ABB RAPID module: 76182c52.mod

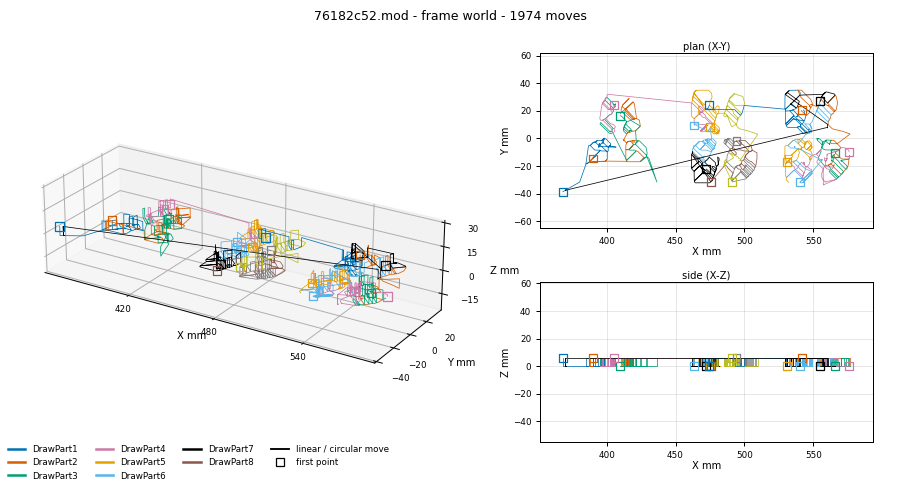
[picture p0: tool path of 76182c52.mod in frame world, 1974 of 1976 moves have a stored position in this frame; points joined in program order, loops and branches not executed]
MODULE ImageDraw
  ! Generated 2026-10-07 06:11 for ABB GoFa CRB 15000-5/0.95: 181 strokes
  ! Page 250 x 180 mm. Work object wPaper: Z points up, so pen-up is +Z and the tool uses orientation [0,1,0,0].
  PERS tooldata tPen:=[TRUE,[[0,0,120],[1,0,0,0]],[0.3,[0,0,60],[1,0,0,0],0,0,0]];
  PERS wobjdata wPaper:=[FALSE,TRUE,"",[[350,-90,0],[1,0,0,0]],[[0,0,0],[1,0,0,0]]];
  CONST robtarget pOrigin:=[[0,0,0],[0,1,0,0],[0,0,0,0],[9E9,9E9,9E9,9E9,9E9,9E9]];
  CONST jointtarget jHome:=[[0,0,0,0,30,0],[9E9,9E9,9E9,9E9,9E9,9E9]];
  CONST speeddata vTravel:=[250,200,5000,1000];

  PROC main()
    SingArea\Wrist;
    ConfL\Off;
    ConfJ\Off;
    MoveAbsJ jHome\NoEOffs,vTravel,fine,tPen;
    DrawPart1;
    DrawPart2;
    DrawPart3;
    DrawPart4;
    DrawPart5;
    DrawPart6;
    DrawPart7;
    DrawPart8;
    DrawPart9;
    DrawPart10;
    DrawPart11;
    DrawPart12;
    DrawPart13;
    DrawPart14;
    DrawPart15;
    DrawPart16;
    DrawPart17;
    MoveAbsJ jHome\NoEOffs,vTravel,fine,tPen;
  ENDPROC

  PROC DrawPart1()
    MoveL Offs(pOrigin,18.35,51.38,6.00),vTravel,z5,tPen\WObj:=wPaper;
    MoveL Offs(pOrigin,18.35,51.38,0.00),v60,z0,tPen\WObj:=wPaper;
    MoveL Offs(pOrigin,30.50,58.42,0.00),v40,z0,tPen\WObj:=wPaper;
    MoveL Offs(pOrigin,35.05,71.47,0.00),v40,z0,tPen\WObj:=wPaper;
    MoveL Offs(pOrigin,37.10,72.53,0.00),v40,z0,tPen\WObj:=wPaper;
    MoveL Offs(pOrigin,37.10,72.53,0.00),v40,z0,tPen\WObj:=wPaper;
    MoveL Offs(pOrigin,38.15,72.53,0.00),v40,z0,tPen\WObj:=wPaper;
    MoveL Offs(pOrigin,39.50,73.12,0.00),v40,z0,tPen\WObj:=wPaper;
    MoveL Offs(pOrigin,48.95,73.28,0.00),v40,z0,tPen\WObj:=wPaper;
    MoveL Offs(pOrigin,50.45,75.07,0.00),v40,z0,tPen\WObj:=wPaper;
    MoveL Offs(pOrigin,50.45,80.03,0.00),v40,z0,tPen\WObj:=wPaper;
    MoveL Offs(pOrigin,51.20,81.07,0.00),v40,z0,tPen\WObj:=wPaper;
    MoveL Offs(pOrigin,51.20,83.47,0.00),v40,z0,tPen\WObj:=wPaper;
    MoveL Offs(pOrigin,51.20,83.47,0.00),v40,z0,tPen\WObj:=wPaper;
    MoveL Offs(pOrigin,47.75,86.78,0.00),v40,z0,tPen\WObj:=wPaper;
    MoveL Offs(pOrigin,47.75,86.78,0.00),v40,z0,tPen\WObj:=wPaper;
    MoveL Offs(pOrigin,47.15,87.53,0.00),v40,z0,tPen\WObj:=wPaper;
    MoveL Offs(pOrigin,47.15,88.43,0.00),v40,z0,tPen\WObj:=wPaper;
    MoveL Offs(pOrigin,47.15,88.43,0.00),v40,z0,tPen\WObj:=wPaper;
    MoveL Offs(pOrigin,48.65,89.93,0.00),v40,z0,tPen\WObj:=wPaper;
    MoveL Offs(pOrigin,48.65,89.93,0.00),v40,z0,tPen\WObj:=wPaper;
    MoveL Offs(pOrigin,47.15,88.43,0.00),v40,z0,tPen\WObj:=wPaper;
    MoveL Offs(pOrigin,46.55,88.57,0.00),v40,z0,tPen\WObj:=wPaper;
    MoveL Offs(pOrigin,48.05,90.07,0.00),v40,fine,tPen\WObj:=wPaper;
    MoveL Offs(pOrigin,48.05,90.07,6.00),v60,z5,tPen\WObj:=wPaper;
    MoveL Offs(pOrigin,47.75,86.78,6.00),vTravel,z5,tPen\WObj:=wPaper;
    MoveL Offs(pOrigin,47.75,86.78,0.00),v60,z0,tPen\WObj:=wPaper;
    MoveL Offs(pOrigin,46.70,86.78,0.00),v40,z0,tPen\WObj:=wPaper;
    MoveL Offs(pOrigin,47.00,86.78,0.00),v40,fine,tPen\WObj:=wPaper;
    MoveL Offs(pOrigin,47.00,86.78,6.00),v60,z5,tPen\WObj:=wPaper;
    MoveL Offs(pOrigin,45.35,85.72,6.00),vTravel,z5,tPen\WObj:=wPaper;
    MoveL Offs(pOrigin,45.35,85.72,0.00),v60,z0,tPen\WObj:=wPaper;
    MoveL Offs(pOrigin,45.35,85.12,0.00),v40,z0,tPen\WObj:=wPaper;
    MoveL Offs(pOrigin,50.45,80.32,0.00),v40,z0,tPen\WObj:=wPaper;
    MoveL Offs(pOrigin,49.55,80.93,0.00),v40,z0,tPen\WObj:=wPaper;
    MoveL Offs(pOrigin,46.55,80.93,0.00),v40,z0,tPen\WObj:=wPaper;
    MoveL Offs(pOrigin,45.35,81.22,0.00),v40,z0,tPen\WObj:=wPaper;
    MoveL Offs(pOrigin,45.35,81.22,0.00),v40,z0,tPen\WObj:=wPaper;
    MoveL Offs(pOrigin,43.10,78.97,0.00),v40,z0,tPen\WObj:=wPaper;
    MoveL Offs(pOrigin,43.10,78.97,0.00),v40,z0,tPen\WObj:=wPaper;
    MoveL Offs(pOrigin,45.35,81.22,0.00),v40,z0,tPen\WObj:=wPaper;
    MoveL Offs(pOrigin,45.35,81.22,0.00),v40,z0,tPen\WObj:=wPaper;
    MoveL Offs(pOrigin,44.75,81.53,0.00),v40,z0,tPen\WObj:=wPaper;
    MoveL Offs(pOrigin,41.45,81.57,0.00),v40,z0,tPen\WObj:=wPaper;
    MoveL Offs(pOrigin,38.15,84.82,0.00),v40,z0,tPen\WObj:=wPaper;
    MoveL Offs(pOrigin,38.15,84.82,0.00),v40,z0,tPen\WObj:=wPaper;
    MoveL Offs(pOrigin,40.55,87.18,0.00),v40,z0,tPen\WObj:=wPaper;
    MoveL Offs(pOrigin,42.05,87.22,0.00),v40,z0,tPen\WObj:=wPaper;
    MoveL Offs(pOrigin,42.05,87.22,0.00),v40,z0,tPen\WObj:=wPaper;
    MoveL Offs(pOrigin,43.40,88.68,0.00),v40,z0,tPen\WObj:=wPaper;
    MoveL Offs(pOrigin,46.25,88.57,0.00),v40,z0,tPen\WObj:=wPaper;
    MoveL Offs(pOrigin,48.35,90.22,0.00),v40,z0,tPen\WObj:=wPaper;
    MoveL Offs(pOrigin,49.55,89.62,0.00),v40,z0,tPen\WObj:=wPaper;
    MoveL Offs(pOrigin,52.85,86.32,0.00),v40,z0,tPen\WObj:=wPaper;
    MoveL Offs(pOrigin,52.85,86.32,0.00),v40,z0,tPen\WObj:=wPaper;
    MoveL Offs(pOrigin,52.80,85.28,0.00),v40,z0,tPen\WObj:=wPaper;
    MoveL Offs(pOrigin,51.20,83.47,0.00),v40,z0,tPen\WObj:=wPaper;
    MoveL Offs(pOrigin,51.65,83.78,0.00),v40,z0,tPen\WObj:=wPaper;
    MoveL Offs(pOrigin,56.75,83.78,0.00),v40,z0,tPen\WObj:=wPaper;
    MoveL Offs(pOrigin,56.45,83.78,0.00),v40,fine,tPen\WObj:=wPaper;
    MoveL Offs(pOrigin,56.45,83.78,6.00),v60,z5,tPen\WObj:=wPaper;
    MoveL Offs(pOrigin,52.10,84.38,6.00),vTravel,z5,tPen\WObj:=wPaper;
    MoveL Offs(pOrigin,52.10,84.38,0.00),v60,z0,tPen\WObj:=wPaper;
    MoveL Offs(pOrigin,52.85,85.12,0.00),v40,z0,tPen\WObj:=wPaper;
    MoveL Offs(pOrigin,52.10,84.38,0.00),v40,fine,tPen\WObj:=wPaper;
    MoveL Offs(pOrigin,52.10,84.38,6.00),v60,z5,tPen\WObj:=wPaper;
    MoveL Offs(pOrigin,46.25,84.07,6.00),vTravel,z5,tPen\WObj:=wPaper;
    MoveL Offs(pOrigin,46.25,84.07,0.00),v60,z0,tPen\WObj:=wPaper;
    MoveL Offs(pOrigin,44.45,84.07,0.00),v40,z0,tPen\WObj:=wPaper;
    MoveL Offs(pOrigin,44.45,84.07,0.00),v40,z0,tPen\WObj:=wPaper;
    MoveL Offs(pOrigin,44.45,83.78,0.00),v40,z0,tPen\WObj:=wPaper;
    MoveL Offs(pOrigin,44.15,83.78,0.00),v40,z0,tPen\WObj:=wPaper;
    MoveL Offs(pOrigin,44.15,84.07,0.00),v40,z0,tPen\WObj:=wPaper;
    MoveL Offs(pOrigin,44.45,84.07,0.00),v40,z0,tPen\WObj:=wPaper;
    MoveL Offs(pOrigin,44.45,83.78,0.00),v40,z0,tPen\WObj:=wPaper;
    MoveL Offs(pOrigin,44.15,83.78,0.00),v40,z0,tPen\WObj:=wPaper;
    MoveL Offs(pOrigin,44.15,84.07,0.00),v40,z0,tPen\WObj:=wPaper;
    MoveL Offs(pOrigin,44.45,84.07,0.00),v40,z0,tPen\WObj:=wPaper;
    MoveL Offs(pOrigin,44.45,84.68,0.00),v40,z0,tPen\WObj:=wPaper;
    MoveL Offs(pOrigin,44.45,84.97,0.00),v40,z0,tPen\WObj:=wPaper;
    MoveL Offs(pOrigin,44.75,84.97,0.00),v40,z0,tPen\WObj:=wPaper;
    MoveL Offs(pOrigin,44.75,84.68,0.00),v40,z0,tPen\WObj:=wPaper;
    MoveL Offs(pOrigin,44.45,84.68,0.00),v40,z0,tPen\WObj:=wPaper;
    MoveL Offs(pOrigin,44.45,84.97,0.00),v40,z0,tPen\WObj:=wPaper;
    MoveL Offs(pOrigin,44.75,84.97,0.00),v40,z0,tPen\WObj:=wPaper;
    MoveL Offs(pOrigin,44.75,84.68,0.00),v40,z0,tPen\WObj:=wPaper;
    MoveL Offs(pOrigin,44.45,84.68,0.00),v40,z0,tPen\WObj:=wPaper;
    MoveL Offs(pOrigin,44.75,84.97,0.00),v40,z0,tPen\WObj:=wPaper;
    MoveL Offs(pOrigin,45.35,85.72,0.00),v40,z0,tPen\WObj:=wPaper;
    MoveL Offs(pOrigin,45.05,86.03,0.00),v40,z0,tPen\WObj:=wPaper;
    MoveL Offs(pOrigin,44.60,86.32,0.00),v40,z0,tPen\WObj:=wPaper;
    MoveL Offs(pOrigin,44.90,85.88,0.00),v40,z0,tPen\WObj:=wPaper;
    MoveL Offs(pOrigin,44.90,85.88,0.00),v40,z0,tPen\WObj:=wPaper;
    MoveL Offs(pOrigin,44.60,85.57,0.00),v40,z0,tPen\WObj:=wPaper;
    MoveL Offs(pOrigin,43.55,85.62,0.00),v40,z0,tPen\WObj:=wPaper;
    MoveL Offs(pOrigin,42.05,87.22,0.00),v40,z0,tPen\WObj:=wPaper;
    MoveL Offs(pOrigin,42.05,87.22,0.00),v40,z0,tPen\WObj:=wPaper;
    MoveL Offs(pOrigin,43.40,88.57,0.00),v40,fine,tPen\WObj:=wPaper;
    MoveL Offs(pOrigin,43.40,88.57,6.00),v60,z5,tPen\WObj:=wPaper;
    MoveL Offs(pOrigin,40.25,87.07,6.00),vTravel,z5,tPen\WObj:=wPaper;
    MoveL Offs(pOrigin,40.25,87.07,0.00),v60,z0,tPen\WObj:=wPaper;
    MoveL Offs(pOrigin,38.15,84.97,0.00),v40,z0,tPen\WObj:=wPaper;
    MoveL Offs(pOrigin,36.85,84.68,0.00),v40,z0,tPen\WObj:=wPaper;
    MoveL Offs(pOrigin,35.00,71.62,0.00),v40,fine,tPen\WObj:=wPaper;
    MoveL Offs(pOrigin,35.00,71.62,6.00),v60,z5,tPen\WObj:=wPaper;
    MoveL Offs(pOrigin,37.10,72.53,6.00),vTravel,z5,tPen\WObj:=wPaper;
    MoveL Offs(pOrigin,37.10,72.53,0.00),v60,z0,tPen\WObj:=wPaper;
    MoveL Offs(pOrigin,41.60,77.47,0.00),v40,z0,tPen\WObj:=wPaper;
    MoveL Offs(pOrigin,41.90,77.47,0.00),v40,z0,tPen\WObj:=wPaper;
    MoveL Offs(pOrigin,42.05,77.03,0.00),v40,z0,tPen\WObj:=wPaper;
    MoveL Offs(pOrigin,41.95,77.78,0.00),v40,z0,tPen\WObj:=wPaper;
    MoveL Offs(pOrigin,42.80,78.68,0.00),v40,z0,tPen\WObj:=wPaper;
    MoveL Offs(pOrigin,42.80,78.68,0.00),v40,z0,tPen\WObj:=wPaper;
    MoveL Offs(pOrigin,41.75,77.78,0.00),v40,z0,tPen\WObj:=wPaper;
    MoveL Offs(pOrigin,41.90,77.47,0.00),v40,fine,tPen\WObj:=wPaper;
    MoveL Offs(pOrigin,41.90,77.47,6.00),v60,z5,tPen\WObj:=wPaper;
    MoveL Offs(pOrigin,39.85,75.47,6.00),vTravel,z5,tPen\WObj:=wPaper;
    MoveL Offs(pOrigin,39.85,75.47,0.00),v60,z0,tPen\WObj:=wPaper;
    MoveL Offs(pOrigin,41.45,77.03,0.00),v40,z0,tPen\WObj:=wPaper;
    MoveL Offs(pOrigin,39.85,75.47,0.00),v40,fine,tPen\WObj:=wPaper;
  ENDPROC

  PROC DrawPart2()
    MoveL Offs(pOrigin,39.85,75.47,6.00),v60,z5,tPen\WObj:=wPaper;
    MoveL Offs(pOrigin,38.05,73.68,6.00),vTravel,z5,tPen\WObj:=wPaper;
    MoveL Offs(pOrigin,38.05,73.68,0.00),v60,z0,tPen\WObj:=wPaper;
    MoveL Offs(pOrigin,39.50,75.07,0.00),v40,z0,tPen\WObj:=wPaper;
    MoveL Offs(pOrigin,38.05,73.68,0.00),v40,z0,tPen\WObj:=wPaper;
    MoveL Offs(pOrigin,37.40,72.97,0.00),v40,z0,tPen\WObj:=wPaper;
    MoveL Offs(pOrigin,37.85,73.43,0.00),v40,z0,tPen\WObj:=wPaper;
    MoveL Offs(pOrigin,37.40,72.97,0.00),v40,fine,tPen\WObj:=wPaper;
    MoveL Offs(pOrigin,37.40,72.97,6.00),v60,z5,tPen\WObj:=wPaper;
    MoveL Offs(pOrigin,49.10,73.57,6.00),vTravel,z5,tPen\WObj:=wPaper;
    MoveL Offs(pOrigin,49.10,73.57,0.00),v60,z0,tPen\WObj:=wPaper;
    MoveL Offs(pOrigin,50.15,74.62,0.00),v40,z0,tPen\WObj:=wPaper;
    MoveL Offs(pOrigin,49.10,73.57,0.00),v40,fine,tPen\WObj:=wPaper;
    MoveL Offs(pOrigin,49.10,73.57,6.00),v60,z5,tPen\WObj:=wPaper;
    MoveL Offs(pOrigin,64.55,73.43,6.00),vTravel,z5,tPen\WObj:=wPaper;
    MoveL Offs(pOrigin,64.55,73.43,0.00),v60,z0,tPen\WObj:=wPaper;
    MoveL Offs(pOrigin,64.85,73.12,0.00),v40,z0,tPen\WObj:=wPaper;
    MoveL Offs(pOrigin,74.15,73.12,0.00),v40,z0,tPen\WObj:=wPaper;
    MoveL Offs(pOrigin,77.10,76.12,0.00),v40,z0,tPen\WObj:=wPaper;
    MoveL Offs(pOrigin,72.50,80.78,0.00),v40,z0,tPen\WObj:=wPaper;
    MoveL Offs(pOrigin,71.60,80.93,0.00),v40,z0,tPen\WObj:=wPaper;
    MoveL Offs(pOrigin,64.70,74.18,0.00),v40,z0,tPen\WObj:=wPaper;
    MoveL Offs(pOrigin,64.55,73.43,0.00),v40,z0,tPen\WObj:=wPaper;
    MoveL Offs(pOrigin,64.55,74.18,0.00),v40,z0,tPen\WObj:=wPaper;
    MoveL Offs(pOrigin,63.95,74.78,0.00),v40,z0,tPen\WObj:=wPaper;
    MoveL Offs(pOrigin,63.95,81.82,0.00),v40,fine,tPen\WObj:=wPaper;
    MoveL Offs(pOrigin,63.95,81.82,6.00),v60,z5,tPen\WObj:=wPaper;
    MoveL Offs(pOrigin,66.20,81.82,6.00),vTravel,z5,tPen\WObj:=wPaper;
    MoveL Offs(pOrigin,66.20,81.82,0.00),v60,z0,tPen\WObj:=wPaper;
    MoveL Offs(pOrigin,68.60,84.22,0.00),v40,fine,tPen\WObj:=wPaper;
    MoveL Offs(pOrigin,68.60,84.22,6.00),v60,z5,tPen\WObj:=wPaper;
    MoveL Offs(pOrigin,69.50,85.57,6.00),vTravel,z5,tPen\WObj:=wPaper;
    MoveL Offs(pOrigin,69.50,85.57,0.00),v60,z0,tPen\WObj:=wPaper;
    MoveL Offs(pOrigin,66.20,81.97,0.00),v40,z0,tPen\WObj:=wPaper;
    MoveL Offs(pOrigin,64.25,81.82,0.00),v40,z0,tPen\WObj:=wPaper;
    MoveL Offs(pOrigin,63.95,82.12,0.00),v40,z0,tPen\WObj:=wPaper;
    MoveL Offs(pOrigin,63.95,85.28,0.00),v40,z0,tPen\WObj:=wPaper;
    MoveL Offs(pOrigin,64.40,86.03,0.00),v40,z0,tPen\WObj:=wPaper;
    MoveL Offs(pOrigin,64.40,86.78,0.00),v40,z0,tPen\WObj:=wPaper;
    MoveL Offs(pOrigin,64.40,86.78,0.00),v40,z0,tPen\WObj:=wPaper;
    MoveL Offs(pOrigin,65.45,87.78,0.00),v40,z0,tPen\WObj:=wPaper;
    MoveL Offs(pOrigin,69.35,88.57,0.00),v40,z0,tPen\WObj:=wPaper;
    MoveL Offs(pOrigin,69.35,88.57,0.00),v40,z0,tPen\WObj:=wPaper;
    MoveL Offs(pOrigin,70.55,87.22,0.00),v40,z0,tPen\WObj:=wPaper;
    MoveL Offs(pOrigin,71.00,86.18,0.00),v40,z0,tPen\WObj:=wPaper;
    MoveL Offs(pOrigin,71.00,86.18,0.00),v40,z0,tPen\WObj:=wPaper;
    MoveL Offs(pOrigin,73.10,88.43,0.00),v40,z0,tPen\WObj:=wPaper;
    MoveL Offs(pOrigin,73.10,88.43,0.00),v40,z0,tPen\WObj:=wPaper;
    MoveL Offs(pOrigin,71.30,88.72,0.00),v40,z0,tPen\WObj:=wPaper;
    MoveL Offs(pOrigin,69.35,88.57,0.00),v40,z0,tPen\WObj:=wPaper;
    MoveL Offs(pOrigin,68.60,88.28,0.00),v40,z0,tPen\WObj:=wPaper;
    MoveL Offs(pOrigin,69.20,87.53,0.00),v40,fine,tPen\WObj:=wPaper;
    MoveL Offs(pOrigin,69.20,87.53,6.00),v60,z5,tPen\WObj:=wPaper;
    MoveL Offs(pOrigin,69.20,86.03,6.00),vTravel,z5,tPen\WObj:=wPaper;
    MoveL Offs(pOrigin,69.20,86.03,0.00),v60,z0,tPen\WObj:=wPaper;
    MoveL Offs(pOrigin,67.55,87.97,0.00),v40,fine,tPen\WObj:=wPaper;
    MoveL Offs(pOrigin,67.55,87.97,6.00),v60,z5,tPen\WObj:=wPaper;
    MoveL Offs(pOrigin,65.45,87.68,6.00),vTravel,z5,tPen\WObj:=wPaper;
    MoveL Offs(pOrigin,65.45,87.68,0.00),v60,z0,tPen\WObj:=wPaper;
    MoveL Offs(pOrigin,64.40,86.78,0.00),v40,z0,tPen\WObj:=wPaper;
    MoveL Offs(pOrigin,64.40,86.78,0.00),v40,z0,tPen\WObj:=wPaper;
    MoveL Offs(pOrigin,62.75,88.43,0.00),v40,z0,tPen\WObj:=wPaper;
    MoveL Offs(pOrigin,62.00,89.03,0.00),v40,z0,tPen\WObj:=wPaper;
    MoveL Offs(pOrigin,62.70,88.57,0.00),v40,z0,tPen\WObj:=wPaper;
    MoveL Offs(pOrigin,62.75,89.78,0.00),v40,fine,tPen\WObj:=wPaper;
    MoveL Offs(pOrigin,62.75,89.78,6.00),v60,z5,tPen\WObj:=wPaper;
    MoveL Offs(pOrigin,65.15,94.12,6.00),vTravel,z5,tPen\WObj:=wPaper;
    MoveL Offs(pOrigin,65.15,94.12,0.00),v60,z0,tPen\WObj:=wPaper;
    MoveL Offs(pOrigin,65.60,94.72,0.00),v40,z0,tPen\WObj:=wPaper;
    MoveL Offs(pOrigin,66.05,94.12,0.00),v40,z0,tPen\WObj:=wPaper;
    MoveL Offs(pOrigin,66.05,94.12,0.00),v40,z0,tPen\WObj:=wPaper;
    MoveL Offs(pOrigin,68.90,95.32,0.00),v40,z0,tPen\WObj:=wPaper;
    MoveL Offs(pOrigin,70.85,95.43,0.00),v40,z0,tPen\WObj:=wPaper;
    MoveL Offs(pOrigin,74.45,98.93,0.00),v40,z0,tPen\WObj:=wPaper;
    MoveL Offs(pOrigin,74.45,98.93,0.00),v40,z0,tPen\WObj:=wPaper;
    MoveL Offs(pOrigin,73.80,103.28,0.00),v40,z0,tPen\WObj:=wPaper;
    MoveL Offs(pOrigin,71.60,104.47,0.00),v40,z0,tPen\WObj:=wPaper;
    MoveL Offs(pOrigin,70.70,104.32,0.00),v40,z0,tPen\WObj:=wPaper;
    MoveL Offs(pOrigin,69.80,104.03,0.00),v40,z0,tPen\WObj:=wPaper;
    MoveL Offs(pOrigin,69.80,104.03,0.00),v40,z0,tPen\WObj:=wPaper;
    MoveL Offs(pOrigin,68.60,104.03,0.00),v40,z0,tPen\WObj:=wPaper;
    MoveL Offs(pOrigin,63.20,109.57,0.00),v40,z0,tPen\WObj:=wPaper;
    MoveL Offs(pOrigin,63.20,109.57,0.00),v40,z0,tPen\WObj:=wPaper;
    MoveL Offs(pOrigin,63.80,110.47,0.00),v40,z0,tPen\WObj:=wPaper;
    MoveL Offs(pOrigin,63.80,110.47,0.00),v40,z0,tPen\WObj:=wPaper;
    MoveL Offs(pOrigin,69.80,104.03,0.00),v40,z0,tPen\WObj:=wPaper;
    MoveL Offs(pOrigin,70.70,104.32,0.00),v40,z0,tPen\WObj:=wPaper;
    MoveL Offs(pOrigin,65.30,109.88,0.00),v40,fine,tPen\WObj:=wPaper;
    MoveL Offs(pOrigin,65.30,109.88,6.00),v60,z5,tPen\WObj:=wPaper;
    MoveL Offs(pOrigin,64.10,111.53,6.00),vTravel,z5,tPen\WObj:=wPaper;
    MoveL Offs(pOrigin,64.10,111.53,0.00),v60,z0,tPen\WObj:=wPaper;
    MoveL Offs(pOrigin,69.20,116.47,0.00),v40,z0,tPen\WObj:=wPaper;
    MoveL Offs(pOrigin,69.20,116.47,0.00),v40,z0,tPen\WObj:=wPaper;
    MoveL Offs(pOrigin,70.10,115.28,0.00),v40,z0,tPen\WObj:=wPaper;
    MoveL Offs(pOrigin,71.60,105.38,0.00),v40,z0,tPen\WObj:=wPaper;
    MoveL Offs(pOrigin,71.45,104.47,0.00),v40,z0,tPen\WObj:=wPaper;
    MoveL Offs(pOrigin,70.70,104.32,0.00),v40,fine,tPen\WObj:=wPaper;
    MoveL Offs(pOrigin,70.70,104.32,6.00),v60,z5,tPen\WObj:=wPaper;
    MoveL Offs(pOrigin,68.60,103.88,6.00),vTravel,z5,tPen\WObj:=wPaper;
    MoveL Offs(pOrigin,68.60,103.88,0.00),v60,z0,tPen\WObj:=wPaper;
    MoveL Offs(pOrigin,68.00,103.32,0.00),v40,z0,tPen\WObj:=wPaper;
    MoveL Offs(pOrigin,67.40,103.43,0.00),v40,z0,tPen\WObj:=wPaper;
    MoveL Offs(pOrigin,60.50,110.03,0.00),v40,z0,tPen\WObj:=wPaper;
    MoveL Offs(pOrigin,60.50,110.03,0.00),v40,z0,tPen\WObj:=wPaper;
    MoveL Offs(pOrigin,60.65,111.68,0.00),v40,z0,tPen\WObj:=wPaper;
    MoveL Offs(pOrigin,61.60,114.22,0.00),v40,z0,tPen\WObj:=wPaper;
    MoveL Offs(pOrigin,66.35,119.03,0.00),v40,z0,tPen\WObj:=wPaper;
    MoveL Offs(pOrigin,66.35,119.03,0.00),v40,z0,tPen\WObj:=wPaper;
    MoveL Offs(pOrigin,61.70,114.22,0.00),v40,fine,tPen\WObj:=wPaper;
    MoveL Offs(pOrigin,61.70,114.22,6.00),v60,z5,tPen\WObj:=wPaper;
    MoveL Offs(pOrigin,61.40,112.88,6.00),vTravel,z5,tPen\WObj:=wPaper;
    MoveL Offs(pOrigin,61.40,112.88,0.00),v60,z0,tPen\WObj:=wPaper;
    MoveL Offs(pOrigin,63.50,111.22,0.00),v40,z0,tPen\WObj:=wPaper;
    MoveL Offs(pOrigin,63.50,111.22,0.00),v40,z0,tPen\WObj:=wPaper;
    MoveL Offs(pOrigin,64.25,111.53,0.00),v40,z0,tPen\WObj:=wPaper;
    MoveL Offs(pOrigin,69.20,116.47,0.00),v40,fine,tPen\WObj:=wPaper;
    MoveL Offs(pOrigin,69.20,116.47,6.00),v60,z5,tPen\WObj:=wPaper;
    MoveL Offs(pOrigin,60.50,108.53,6.00),vTravel,z5,tPen\WObj:=wPaper;
    MoveL Offs(pOrigin,60.50,108.53,0.00),v60,z0,tPen\WObj:=wPaper;
    MoveL Offs(pOrigin,59.90,107.93,0.00),v40,z0,tPen\WObj:=wPaper;
  ENDPROC

  PROC DrawPart3()
    MoveL Offs(pOrigin,59.90,106.57,0.00),v40,z0,tPen\WObj:=wPaper;
    MoveL Offs(pOrigin,59.90,106.57,0.00),v40,z0,tPen\WObj:=wPaper;
    MoveL Offs(pOrigin,60.65,106.28,0.00),v40,z0,tPen\WObj:=wPaper;
    MoveL Offs(pOrigin,64.55,102.38,0.00),v40,z0,tPen\WObj:=wPaper;
    MoveL Offs(pOrigin,64.55,102.38,0.00),v40,z0,tPen\WObj:=wPaper;
    MoveL Offs(pOrigin,63.90,100.43,0.00),v40,z0,tPen\WObj:=wPaper;
    MoveL Offs(pOrigin,62.95,99.38,0.00),v40,z0,tPen\WObj:=wPaper;
    MoveL Offs(pOrigin,62.50,98.18,0.00),v40,z0,tPen\WObj:=wPaper;
    MoveL Offs(pOrigin,62.15,95.62,0.00),v40,z0,tPen\WObj:=wPaper;
    MoveL Offs(pOrigin,64.10,93.57,0.00),v40,z0,tPen\WObj:=wPaper;
    MoveL Offs(pOrigin,64.80,93.57,0.00),v40,z0,tPen\WObj:=wPaper;
    MoveL Offs(pOrigin,65.15,94.12,0.00),v40,z0,tPen\WObj:=wPaper;
    MoveL Offs(pOrigin,65.30,94.28,0.00),v40,z0,tPen\WObj:=wPaper;
    MoveL Offs(pOrigin,62.45,96.97,0.00),v40,fine,tPen\WObj:=wPaper;
    MoveL Offs(pOrigin,62.45,96.97,6.00),v60,z5,tPen\WObj:=wPaper;
    MoveL Offs(pOrigin,62.90,98.47,6.00),vTravel,z5,tPen\WObj:=wPaper;
    MoveL Offs(pOrigin,62.90,98.47,0.00),v60,z0,tPen\WObj:=wPaper;
    MoveL Offs(pOrigin,66.80,94.43,0.00),v40,fine,tPen\WObj:=wPaper;
    MoveL Offs(pOrigin,66.80,94.43,6.00),v60,z5,tPen\WObj:=wPaper;
    MoveL Offs(pOrigin,66.65,95.62,6.00),vTravel,z5,tPen\WObj:=wPaper;
    MoveL Offs(pOrigin,66.65,95.62,0.00),v60,z0,tPen\WObj:=wPaper;
    MoveL Offs(pOrigin,66.80,95.32,0.00),v40,z0,tPen\WObj:=wPaper;
    MoveL Offs(pOrigin,67.10,95.47,0.00),v40,z0,tPen\WObj:=wPaper;
    MoveL Offs(pOrigin,66.80,95.78,0.00),v40,fine,tPen\WObj:=wPaper;
    MoveL Offs(pOrigin,66.80,95.78,6.00),v60,z5,tPen\WObj:=wPaper;
    MoveL Offs(pOrigin,68.60,95.32,6.00),vTravel,z5,tPen\WObj:=wPaper;
    MoveL Offs(pOrigin,68.60,95.32,0.00),v60,z0,tPen\WObj:=wPaper;
    MoveL Offs(pOrigin,67.25,97.12,0.00),v40,z0,tPen\WObj:=wPaper;
    MoveL Offs(pOrigin,63.95,100.28,0.00),v40,z0,tPen\WObj:=wPaper;
    MoveL Offs(pOrigin,63.95,100.28,0.00),v40,z0,tPen\WObj:=wPaper;
    MoveL Offs(pOrigin,63.05,99.38,0.00),v40,fine,tPen\WObj:=wPaper;
    MoveL Offs(pOrigin,63.05,99.38,6.00),v60,z5,tPen\WObj:=wPaper;
    MoveL Offs(pOrigin,64.55,102.38,6.00),vTravel,z5,tPen\WObj:=wPaper;
    MoveL Offs(pOrigin,64.55,102.38,0.00),v60,z0,tPen\WObj:=wPaper;
    MoveL Offs(pOrigin,65.60,102.38,0.00),v40,z0,tPen\WObj:=wPaper;
    MoveL Offs(pOrigin,67.40,103.28,0.00),v40,fine,tPen\WObj:=wPaper;
    MoveL Offs(pOrigin,67.40,103.28,6.00),v60,z5,tPen\WObj:=wPaper;
    MoveL Offs(pOrigin,74.45,98.93,6.00),vTravel,z5,tPen\WObj:=wPaper;
    MoveL Offs(pOrigin,74.45,98.93,0.00),v60,z0,tPen\WObj:=wPaper;
    MoveL Offs(pOrigin,71.00,95.62,0.00),v40,fine,tPen\WObj:=wPaper;
    MoveL Offs(pOrigin,71.00,95.62,6.00),v60,z5,tPen\WObj:=wPaper;
    MoveL Offs(pOrigin,71.60,86.78,6.00),vTravel,z5,tPen\WObj:=wPaper;
    MoveL Offs(pOrigin,71.60,86.78,0.00),v60,z0,tPen\WObj:=wPaper;
    MoveL Offs(pOrigin,73.10,88.28,0.00),v40,z0,tPen\WObj:=wPaper;
    MoveL Offs(pOrigin,73.70,88.38,0.00),v40,z0,tPen\WObj:=wPaper;
    MoveL Offs(pOrigin,78.65,83.47,0.00),v40,z0,tPen\WObj:=wPaper;
    MoveL Offs(pOrigin,79.40,79.43,0.00),v40,z0,tPen\WObj:=wPaper;
    MoveL Offs(pOrigin,79.35,78.53,0.00),v40,z0,tPen\WObj:=wPaper;
    MoveL Offs(pOrigin,78.80,77.93,0.00),v40,z0,tPen\WObj:=wPaper;
    MoveL Offs(pOrigin,78.80,77.93,0.00),v40,z0,tPen\WObj:=wPaper;
    MoveL Offs(pOrigin,78.80,76.72,0.00),v40,z0,tPen\WObj:=wPaper;
    MoveL Offs(pOrigin,78.20,76.18,0.00),v40,z0,tPen\WObj:=wPaper;
    MoveL Offs(pOrigin,77.15,75.97,0.00),v40,z0,tPen\WObj:=wPaper;
    MoveL Offs(pOrigin,77.15,75.97,0.00),v40,z0,tPen\WObj:=wPaper;
    MoveL Offs(pOrigin,74.60,73.28,0.00),v40,fine,tPen\WObj:=wPaper;
    MoveL Offs(pOrigin,74.60,73.28,6.00),v60,z5,tPen\WObj:=wPaper;
    MoveL Offs(pOrigin,78.95,76.72,6.00),vTravel,z5,tPen\WObj:=wPaper;
    MoveL Offs(pOrigin,78.95,76.72,0.00),v60,z0,tPen\WObj:=wPaper;
    MoveL Offs(pOrigin,80.60,75.82,0.00),v40,z0,tPen\WObj:=wPaper;
    MoveL Offs(pOrigin,86.45,58.42,0.00),v40,fine,tPen\WObj:=wPaper;
    MoveL Offs(pOrigin,86.45,58.42,6.00),v60,z5,tPen\WObj:=wPaper;
    MoveL Offs(pOrigin,78.80,77.93,6.00),vTravel,z5,tPen\WObj:=wPaper;
    MoveL Offs(pOrigin,78.80,77.93,0.00),v60,z0,tPen\WObj:=wPaper;
    MoveL Offs(pOrigin,71.15,85.57,0.00),v40,z0,tPen\WObj:=wPaper;
    MoveL Offs(pOrigin,71.00,86.18,0.00),v40,z0,tPen\WObj:=wPaper;
    MoveL Offs(pOrigin,71.00,85.57,0.00),v40,z0,tPen\WObj:=wPaper;
    MoveL Offs(pOrigin,69.50,85.72,0.00),v40,fine,tPen\WObj:=wPaper;
    MoveL Offs(pOrigin,69.50,85.72,6.00),v60,z5,tPen\WObj:=wPaper;
    MoveL Offs(pOrigin,66.20,81.82,6.00),vTravel,z5,tPen\WObj:=wPaper;
    MoveL Offs(pOrigin,66.20,81.82,0.00),v60,z0,tPen\WObj:=wPaper;
    MoveL Offs(pOrigin,66.80,81.53,0.00),v40,z0,tPen\WObj:=wPaper;
    MoveL Offs(pOrigin,70.55,81.53,0.00),v40,z0,tPen\WObj:=wPaper;
    MoveL Offs(pOrigin,71.30,80.93,0.00),v40,z0,tPen\WObj:=wPaper;
    MoveL Offs(pOrigin,71.30,80.93,0.00),v40,z0,tPen\WObj:=wPaper;
    MoveL Offs(pOrigin,64.55,74.18,0.00),v40,fine,tPen\WObj:=wPaper;
    MoveL Offs(pOrigin,64.55,74.18,6.00),v60,z5,tPen\WObj:=wPaper;
    MoveL Offs(pOrigin,54.35,94.43,6.00),vTravel,z5,tPen\WObj:=wPaper;
    MoveL Offs(pOrigin,54.35,94.43,0.00),v60,z0,tPen\WObj:=wPaper;
    MoveL Offs(pOrigin,53.60,93.68,0.00),v40,z0,tPen\WObj:=wPaper;
    MoveL Offs(pOrigin,52.10,93.72,0.00),v40,z0,tPen\WObj:=wPaper;
    MoveL Offs(pOrigin,45.20,100.43,0.00),v40,fine,tPen\WObj:=wPaper;
    MoveL Offs(pOrigin,45.20,100.43,6.00),v60,z5,tPen\WObj:=wPaper;
    MoveL Offs(pOrigin,45.65,101.62,6.00),vTravel,z5,tPen\WObj:=wPaper;
    MoveL Offs(pOrigin,45.65,101.62,0.00),v60,z0,tPen\WObj:=wPaper;
    MoveL Offs(pOrigin,52.25,95.18,0.00),v40,z0,tPen\WObj:=wPaper;
    MoveL Offs(pOrigin,52.55,95.32,0.00),v40,z0,tPen\WObj:=wPaper;
    MoveL Offs(pOrigin,52.55,94.72,0.00),v40,z0,tPen\WObj:=wPaper;
    MoveL Offs(pOrigin,52.85,95.32,0.00),v40,z0,tPen\WObj:=wPaper;
    MoveL Offs(pOrigin,54.05,95.03,0.00),v40,z0,tPen\WObj:=wPaper;
    MoveL Offs(pOrigin,54.05,95.03,0.00),v40,z0,tPen\WObj:=wPaper;
    MoveL Offs(pOrigin,53.90,96.68,0.00),v40,z0,tPen\WObj:=wPaper;
    MoveL Offs(pOrigin,53.90,96.68,0.00),v40,z0,tPen\WObj:=wPaper;
    MoveL Offs(pOrigin,54.95,97.12,0.00),v40,z0,tPen\WObj:=wPaper;
    MoveL Offs(pOrigin,54.95,97.12,0.00),v40,z0,tPen\WObj:=wPaper;
    MoveL Offs(pOrigin,48.50,103.88,0.00),v40,z0,tPen\WObj:=wPaper;
    MoveL Offs(pOrigin,48.50,103.88,0.00),v40,z0,tPen\WObj:=wPaper;
    MoveL Offs(pOrigin,52.10,107.18,0.00),v40,fine,tPen\WObj:=wPaper;
    MoveL Offs(pOrigin,52.10,107.18,6.00),v60,z5,tPen\WObj:=wPaper;
    MoveL Offs(pOrigin,53.45,107.62,6.00),vTravel,z5,tPen\WObj:=wPaper;
    MoveL Offs(pOrigin,53.45,107.62,0.00),v60,z0,tPen\WObj:=wPaper;
    MoveL Offs(pOrigin,54.85,109.57,0.00),v40,z0,tPen\WObj:=wPaper;
    MoveL Offs(pOrigin,54.95,111.82,0.00),v40,z0,tPen\WObj:=wPaper;
    MoveL Offs(pOrigin,54.95,111.82,0.00),v40,z0,tPen\WObj:=wPaper;
    MoveL Offs(pOrigin,48.80,117.82,0.00),v40,z0,tPen\WObj:=wPaper;
    MoveL Offs(pOrigin,48.80,117.82,0.00),v40,z0,tPen\WObj:=wPaper;
    MoveL Offs(pOrigin,49.05,119.18,0.00),v40,z0,tPen\WObj:=wPaper;
    MoveL Offs(pOrigin,50.15,119.93,0.00),v40,z0,tPen\WObj:=wPaper;
    MoveL Offs(pOrigin,50.15,119.93,0.00),v40,z0,tPen\WObj:=wPaper;
    MoveL Offs(pOrigin,54.65,115.43,0.00),v40,z0,tPen\WObj:=wPaper;
    MoveL Offs(pOrigin,54.70,114.72,0.00),v40,z0,tPen\WObj:=wPaper;
    MoveL Offs(pOrigin,54.95,114.97,0.00),v40,z0,tPen\WObj:=wPaper;
    MoveL Offs(pOrigin,54.95,114.97,0.00),v40,z0,tPen\WObj:=wPaper;
    MoveL Offs(pOrigin,55.70,114.38,0.00),v40,z0,tPen\WObj:=wPaper;
    MoveL Offs(pOrigin,56.45,114.57,0.00),v40,z0,tPen\WObj:=wPaper;
    MoveL Offs(pOrigin,56.60,115.12,0.00),v40,z0,tPen\WObj:=wPaper;
    MoveL Offs(pOrigin,56.00,114.38,0.00),v40,z0,tPen\WObj:=wPaper;
    MoveL Offs(pOrigin,56.45,113.47,0.00),v40,z0,tPen\WObj:=wPaper;
    MoveL Offs(pOrigin,55.40,112.43,0.00),v40,z0,tPen\WObj:=wPaper;
    MoveL Offs(pOrigin,55.40,112.43,0.00),v40,z0,tPen\WObj:=wPaper;
    MoveL Offs(pOrigin,55.40,114.38,0.00),v40,fine,tPen\WObj:=wPaper;
  ENDPROC

  PROC DrawPart4()
    MoveL Offs(pOrigin,55.40,114.38,6.00),v60,z5,tPen\WObj:=wPaper;
    MoveL Offs(pOrigin,55.70,112.43,6.00),vTravel,z5,tPen\WObj:=wPaper;
    MoveL Offs(pOrigin,55.70,112.43,0.00),v60,z0,tPen\WObj:=wPaper;
    MoveL Offs(pOrigin,56.45,113.18,0.00),v40,z0,tPen\WObj:=wPaper;
    MoveL Offs(pOrigin,55.70,112.43,0.00),v40,fine,tPen\WObj:=wPaper;
    MoveL Offs(pOrigin,55.70,112.43,6.00),v60,z5,tPen\WObj:=wPaper;
    MoveL Offs(pOrigin,52.40,111.22,6.00),vTravel,z5,tPen\WObj:=wPaper;
    MoveL Offs(pOrigin,52.40,111.22,0.00),v60,z0,tPen\WObj:=wPaper;
    MoveL Offs(pOrigin,54.20,109.12,0.00),v40,fine,tPen\WObj:=wPaper;
    MoveL Offs(pOrigin,54.20,109.12,6.00),v60,z5,tPen\WObj:=wPaper;
    MoveL Offs(pOrigin,53.45,107.62,6.00),vTravel,z5,tPen\WObj:=wPaper;
    MoveL Offs(pOrigin,53.45,107.62,0.00),v60,z0,tPen\WObj:=wPaper;
    MoveL Offs(pOrigin,52.25,107.18,0.00),v40,z0,tPen\WObj:=wPaper;
    MoveL Offs(pOrigin,49.40,104.32,0.00),v40,z0,tPen\WObj:=wPaper;
    MoveL Offs(pOrigin,49.40,104.32,0.00),v40,z0,tPen\WObj:=wPaper;
    MoveL Offs(pOrigin,52.70,100.88,0.00),v40,z0,tPen\WObj:=wPaper;
    MoveL Offs(pOrigin,54.95,100.12,0.00),v40,z0,tPen\WObj:=wPaper;
    MoveL Offs(pOrigin,56.20,98.78,0.00),v40,z0,tPen\WObj:=wPaper;
    MoveL Offs(pOrigin,56.30,98.03,0.00),v40,z0,tPen\WObj:=wPaper;
    MoveL Offs(pOrigin,56.30,98.03,0.00),v40,z0,tPen\WObj:=wPaper;
    MoveL Offs(pOrigin,55.40,97.12,0.00),v40,z0,tPen\WObj:=wPaper;
    MoveL Offs(pOrigin,55.40,97.12,0.00),v40,z0,tPen\WObj:=wPaper;
    MoveL Offs(pOrigin,55.95,95.18,0.00),v40,z0,tPen\WObj:=wPaper;
    MoveL Offs(pOrigin,55.10,94.43,0.00),v40,z0,tPen\WObj:=wPaper;
    MoveL Offs(pOrigin,54.50,94.47,0.00),v40,z0,tPen\WObj:=wPaper;
    MoveL Offs(pOrigin,54.05,95.03,0.00),v40,fine,tPen\WObj:=wPaper;
    MoveL Offs(pOrigin,54.05,95.03,6.00),v60,z5,tPen\WObj:=wPaper;
    MoveL Offs(pOrigin,53.90,96.68,6.00),vTravel,z5,tPen\WObj:=wPaper;
    MoveL Offs(pOrigin,53.90,96.68,0.00),v60,z0,tPen\WObj:=wPaper;
    MoveL Offs(pOrigin,47.15,103.28,0.00),v40,z0,tPen\WObj:=wPaper;
    MoveL Offs(pOrigin,47.15,103.28,0.00),v40,z0,tPen\WObj:=wPaper;
    MoveL Offs(pOrigin,47.75,103.88,0.00),v40,z0,tPen\WObj:=wPaper;
    MoveL Offs(pOrigin,48.50,103.88,0.00),v40,fine,tPen\WObj:=wPaper;
    MoveL Offs(pOrigin,48.50,103.88,6.00),v60,z5,tPen\WObj:=wPaper;
    MoveL Offs(pOrigin,47.15,103.28,6.00),vTravel,z5,tPen\WObj:=wPaper;
    MoveL Offs(pOrigin,47.15,103.28,0.00),v60,z0,tPen\WObj:=wPaper;
    MoveL Offs(pOrigin,45.80,103.12,0.00),v40,z0,tPen\WObj:=wPaper;
    MoveL Offs(pOrigin,45.80,103.12,0.00),v40,z0,tPen\WObj:=wPaper;
    MoveL Offs(pOrigin,45.05,104.32,0.00),v40,z0,tPen\WObj:=wPaper;
    MoveL Offs(pOrigin,46.55,114.38,0.00),v40,z0,tPen\WObj:=wPaper;
    MoveL Offs(pOrigin,47.00,115.12,0.00),v40,z0,tPen\WObj:=wPaper;
    MoveL Offs(pOrigin,47.00,115.12,0.00),v40,z0,tPen\WObj:=wPaper;
    MoveL Offs(pOrigin,51.20,111.07,0.00),v40,z0,tPen\WObj:=wPaper;
    MoveL Offs(pOrigin,51.20,111.07,0.00),v40,z0,tPen\WObj:=wPaper;
    MoveL Offs(pOrigin,51.50,111.07,0.00),v40,z0,tPen\WObj:=wPaper;
    MoveL Offs(pOrigin,51.35,110.78,0.00),v40,z0,tPen\WObj:=wPaper;
    MoveL Offs(pOrigin,51.20,111.07,0.00),v40,z0,tPen\WObj:=wPaper;
    MoveL Offs(pOrigin,51.50,111.07,0.00),v40,z0,tPen\WObj:=wPaper;
    MoveL Offs(pOrigin,51.20,110.78,0.00),v40,z0,tPen\WObj:=wPaper;
    MoveL Offs(pOrigin,51.20,111.07,0.00),v40,fine,tPen\WObj:=wPaper;
    MoveL Offs(pOrigin,51.20,111.07,6.00),v60,z5,tPen\WObj:=wPaper;
    MoveL Offs(pOrigin,52.40,111.22,6.00),vTravel,z5,tPen\WObj:=wPaper;
    MoveL Offs(pOrigin,52.40,111.22,0.00),v60,z0,tPen\WObj:=wPaper;
    MoveL Offs(pOrigin,47.45,116.03,0.00),v40,z0,tPen\WObj:=wPaper;
    MoveL Offs(pOrigin,47.45,116.03,0.00),v40,z0,tPen\WObj:=wPaper;
    MoveL Offs(pOrigin,47.75,117.07,0.00),v40,z0,tPen\WObj:=wPaper;
    MoveL Offs(pOrigin,48.80,117.82,0.00),v40,fine,tPen\WObj:=wPaper;
    MoveL Offs(pOrigin,48.80,117.82,6.00),v60,z5,tPen\WObj:=wPaper;
    MoveL Offs(pOrigin,47.45,116.03,6.00),vTravel,z5,tPen\WObj:=wPaper;
    MoveL Offs(pOrigin,47.45,116.03,0.00),v60,z0,tPen\WObj:=wPaper;
    MoveL Offs(pOrigin,47.00,115.72,0.00),v40,z0,tPen\WObj:=wPaper;
    MoveL Offs(pOrigin,47.00,115.12,0.00),v40,fine,tPen\WObj:=wPaper;
    MoveL Offs(pOrigin,47.00,115.12,6.00),v60,z5,tPen\WObj:=wPaper;
    MoveL Offs(pOrigin,50.15,119.93,6.00),vTravel,z5,tPen\WObj:=wPaper;
    MoveL Offs(pOrigin,50.15,119.93,0.00),v60,z0,tPen\WObj:=wPaper;
    MoveL Offs(pOrigin,50.35,121.72,0.00),v40,z0,tPen\WObj:=wPaper;
    MoveL Offs(pOrigin,50.90,122.03,0.00),v40,fine,tPen\WObj:=wPaper;
    MoveL Offs(pOrigin,50.90,122.03,6.00),v60,z5,tPen\WObj:=wPaper;
    MoveL Offs(pOrigin,111.95,115.72,6.00),vTravel,z5,tPen\WObj:=wPaper;
    MoveL Offs(pOrigin,111.95,115.72,0.00),v60,z0,tPen\WObj:=wPaper;
    MoveL Offs(pOrigin,118.85,108.97,0.00),v40,z0,tPen\WObj:=wPaper;
    MoveL Offs(pOrigin,119.45,108.97,0.00),v40,z0,tPen\WObj:=wPaper;
    MoveL Offs(pOrigin,121.40,107.03,0.00),v40,z0,tPen\WObj:=wPaper;
    MoveL Offs(pOrigin,122.00,105.68,0.00),v40,z0,tPen\WObj:=wPaper;
    MoveL Offs(pOrigin,127.25,100.72,0.00),v40,z0,tPen\WObj:=wPaper;
    MoveL Offs(pOrigin,127.25,100.72,0.00),v40,z0,tPen\WObj:=wPaper;
    MoveL Offs(pOrigin,126.95,99.97,0.00),v40,z0,tPen\WObj:=wPaper;
    MoveL Offs(pOrigin,126.50,99.97,0.00),v40,z0,tPen\WObj:=wPaper;
    MoveL Offs(pOrigin,126.50,99.97,0.00),v40,z0,tPen\WObj:=wPaper;
    MoveL Offs(pOrigin,121.25,105.03,0.00),v40,z0,tPen\WObj:=wPaper;
    MoveL Offs(pOrigin,119.60,105.53,0.00),v40,z0,tPen\WObj:=wPaper;
    MoveL Offs(pOrigin,117.65,107.62,0.00),v40,z0,tPen\WObj:=wPaper;
    MoveL Offs(pOrigin,117.65,107.62,0.00),v40,z0,tPen\WObj:=wPaper;
    MoveL Offs(pOrigin,118.10,108.68,0.00),v40,z0,tPen\WObj:=wPaper;
    MoveL Offs(pOrigin,118.10,108.68,0.00),v40,z0,tPen\WObj:=wPaper;
    MoveL Offs(pOrigin,119.45,108.97,0.00),v40,z0,tPen\WObj:=wPaper;
    MoveL Offs(pOrigin,119.90,109.72,0.00),v40,z0,tPen\WObj:=wPaper;
    MoveL Offs(pOrigin,120.80,110.18,0.00),v40,z0,tPen\WObj:=wPaper;
    MoveL Offs(pOrigin,120.80,110.62,0.00),v40,z0,tPen\WObj:=wPaper;
    MoveL Offs(pOrigin,118.50,112.97,0.00),v40,z0,tPen\WObj:=wPaper;
    MoveL Offs(pOrigin,117.20,113.47,0.00),v40,z0,tPen\WObj:=wPaper;
    MoveL Offs(pOrigin,117.20,113.47,0.00),v40,z0,tPen\WObj:=wPaper;
    MoveL Offs(pOrigin,117.80,111.82,0.00),v40,z0,tPen\WObj:=wPaper;
    MoveL Offs(pOrigin,119.90,109.72,0.00),v40,fine,tPen\WObj:=wPaper;
    MoveL Offs(pOrigin,119.90,109.72,6.00),v60,z5,tPen\WObj:=wPaper;
    MoveL Offs(pOrigin,118.10,108.68,6.00),vTravel,z5,tPen\WObj:=wPaper;
    MoveL Offs(pOrigin,118.10,108.68,0.00),v60,z0,tPen\WObj:=wPaper;
    MoveL Offs(pOrigin,116.90,109.88,0.00),v40,fine,tPen\WObj:=wPaper;
    MoveL Offs(pOrigin,116.90,109.88,6.00),v60,z5,tPen\WObj:=wPaper;
    MoveL Offs(pOrigin,117.65,107.62,6.00),vTravel,z5,tPen\WObj:=wPaper;
    MoveL Offs(pOrigin,117.65,107.62,0.00),v60,z0,tPen\WObj:=wPaper;
    MoveL Offs(pOrigin,116.45,107.18,0.00),v40,z0,tPen\WObj:=wPaper;
    MoveL Offs(pOrigin,113.50,104.18,0.00),v40,z0,tPen\WObj:=wPaper;
    MoveL Offs(pOrigin,113.50,100.57,0.00),v40,z0,tPen\WObj:=wPaper;
    MoveL Offs(pOrigin,122.60,99.97,0.00),v40,z0,tPen\WObj:=wPaper;
    MoveL Offs(pOrigin,122.60,99.97,0.00),v40,z0,tPen\WObj:=wPaper;
    MoveL Offs(pOrigin,120.50,97.88,0.00),v40,z0,tPen\WObj:=wPaper;
    MoveL Offs(pOrigin,120.05,97.57,0.00),v40,z0,tPen\WObj:=wPaper;
    MoveL Offs(pOrigin,117.95,95.32,0.00),v40,z0,tPen\WObj:=wPaper;
    MoveL Offs(pOrigin,117.95,95.32,0.00),v40,z0,tPen\WObj:=wPaper;
    MoveL Offs(pOrigin,122.60,99.82,0.00),v40,z0,tPen\WObj:=wPaper;
    MoveL Offs(pOrigin,123.05,99.68,0.00),v40,z0,tPen\WObj:=wPaper;
    MoveL Offs(pOrigin,123.05,99.68,0.00),v40,z0,tPen\WObj:=wPaper;
    MoveL Offs(pOrigin,118.70,95.18,0.00),v40,z0,tPen\WObj:=wPaper;
    MoveL Offs(pOrigin,118.70,95.18,0.00),v40,z0,tPen\WObj:=wPaper;
    MoveL Offs(pOrigin,120.50,96.97,0.00),v40,z0,tPen\WObj:=wPaper;
    MoveL Offs(pOrigin,120.80,97.28,0.00),v40,z0,tPen\WObj:=wPaper;
    MoveL Offs(pOrigin,123.05,99.68,0.00),v40,z0,tPen\WObj:=wPaper;
    MoveL Offs(pOrigin,123.05,99.68,0.00),v40,z0,tPen\WObj:=wPaper;
    MoveL Offs(pOrigin,123.80,99.62,0.00),v40,z0,tPen\WObj:=wPaper;
  ENDPROC

  PROC DrawPart5()
    MoveL Offs(pOrigin,125.15,98.32,0.00),v40,z0,tPen\WObj:=wPaper;
    MoveL Offs(pOrigin,125.60,98.32,0.00),v40,z0,tPen\WObj:=wPaper;
    MoveL Offs(pOrigin,125.90,98.93,0.00),v40,z0,tPen\WObj:=wPaper;
    MoveL Offs(pOrigin,126.50,99.07,0.00),v40,z0,tPen\WObj:=wPaper;
    MoveL Offs(pOrigin,126.50,99.07,0.00),v40,z0,tPen\WObj:=wPaper;
    MoveL Offs(pOrigin,126.50,99.97,0.00),v40,z0,tPen\WObj:=wPaper;
    MoveL Offs(pOrigin,127.25,100.12,0.00),v40,z0,tPen\WObj:=wPaper;
    MoveL Offs(pOrigin,131.30,95.93,0.00),v40,z0,tPen\WObj:=wPaper;
    MoveL Offs(pOrigin,131.60,95.93,0.00),v40,z0,tPen\WObj:=wPaper;
    MoveL Offs(pOrigin,131.90,95.03,0.00),v40,z0,tPen\WObj:=wPaper;
    MoveL Offs(pOrigin,131.45,94.57,0.00),v40,z0,tPen\WObj:=wPaper;
    MoveL Offs(pOrigin,131.45,94.57,0.00),v40,z0,tPen\WObj:=wPaper;
    MoveL Offs(pOrigin,131.30,93.43,0.00),v40,z0,tPen\WObj:=wPaper;
    MoveL Offs(pOrigin,129.80,93.22,0.00),v40,z0,tPen\WObj:=wPaper;
    MoveL Offs(pOrigin,128.75,93.53,0.00),v40,z0,tPen\WObj:=wPaper;
    MoveL Offs(pOrigin,128.75,93.53,0.00),v40,z0,tPen\WObj:=wPaper;
    MoveL Offs(pOrigin,128.60,94.28,0.00),v40,z0,tPen\WObj:=wPaper;
    MoveL Offs(pOrigin,125.20,97.72,0.00),v40,z0,tPen\WObj:=wPaper;
    MoveL Offs(pOrigin,125.20,98.18,0.00),v40,z0,tPen\WObj:=wPaper;
    MoveL Offs(pOrigin,125.60,98.32,0.00),v40,z0,tPen\WObj:=wPaper;
    MoveL Offs(pOrigin,125.60,98.32,0.00),v40,z0,tPen\WObj:=wPaper;
    MoveL Offs(pOrigin,129.35,94.57,0.00),v40,z0,tPen\WObj:=wPaper;
    MoveL Offs(pOrigin,129.95,94.43,0.00),v40,z0,tPen\WObj:=wPaper;
    MoveL Offs(pOrigin,130.40,93.82,0.00),v40,z0,tPen\WObj:=wPaper;
    MoveL Offs(pOrigin,131.45,94.57,0.00),v40,z0,tPen\WObj:=wPaper;
    MoveL Offs(pOrigin,131.15,94.57,0.00),v40,z0,tPen\WObj:=wPaper;
    MoveL Offs(pOrigin,130.70,95.03,0.00),v40,z0,tPen\WObj:=wPaper;
    MoveL Offs(pOrigin,131.60,95.93,0.00),v40,z0,tPen\WObj:=wPaper;
    MoveL Offs(pOrigin,131.60,95.93,0.00),v40,z0,tPen\WObj:=wPaper;
    MoveL Offs(pOrigin,131.90,96.38,0.00),v40,z0,tPen\WObj:=wPaper;
    MoveL Offs(pOrigin,131.85,97.57,0.00),v40,z0,tPen\WObj:=wPaper;
    MoveL Offs(pOrigin,128.15,101.32,0.00),v40,z0,tPen\WObj:=wPaper;
    MoveL Offs(pOrigin,128.15,101.32,0.00),v40,z0,tPen\WObj:=wPaper;
    MoveL Offs(pOrigin,129.05,103.72,0.00),v40,z0,tPen\WObj:=wPaper;
    MoveL Offs(pOrigin,129.05,104.62,0.00),v40,z0,tPen\WObj:=wPaper;
    MoveL Offs(pOrigin,129.05,104.62,0.00),v40,z0,tPen\WObj:=wPaper;
    MoveL Offs(pOrigin,129.50,105.22,0.00),v40,z0,tPen\WObj:=wPaper;
    MoveL Offs(pOrigin,129.80,107.18,0.00),v40,z0,tPen\WObj:=wPaper;
    MoveL Offs(pOrigin,129.80,107.18,0.00),v40,z0,tPen\WObj:=wPaper;
    MoveL Offs(pOrigin,130.95,108.22,0.00),v40,z0,tPen\WObj:=wPaper;
    MoveL Offs(pOrigin,131.60,111.82,0.00),v40,z0,tPen\WObj:=wPaper;
    MoveL Offs(pOrigin,131.55,113.12,0.00),v40,z0,tPen\WObj:=wPaper;
    MoveL Offs(pOrigin,130.55,113.78,0.00),v40,fine,tPen\WObj:=wPaper;
    MoveL Offs(pOrigin,130.55,113.78,6.00),v60,z5,tPen\WObj:=wPaper;
    MoveL Offs(pOrigin,126.95,109.88,6.00),vTravel,z5,tPen\WObj:=wPaper;
    MoveL Offs(pOrigin,126.95,109.88,0.00),v60,z0,tPen\WObj:=wPaper;
    MoveL Offs(pOrigin,129.30,107.93,0.00),v40,z0,tPen\WObj:=wPaper;
    MoveL Offs(pOrigin,129.35,109.28,0.00),v40,z0,tPen\WObj:=wPaper;
    MoveL Offs(pOrigin,129.05,109.88,0.00),v40,z0,tPen\WObj:=wPaper;
    MoveL Offs(pOrigin,124.55,114.07,0.00),v40,z0,tPen\WObj:=wPaper;
    MoveL Offs(pOrigin,124.55,114.07,0.00),v40,z0,tPen\WObj:=wPaper;
    MoveL Offs(pOrigin,125.10,116.62,0.00),v40,z0,tPen\WObj:=wPaper;
    MoveL Offs(pOrigin,125.60,117.07,0.00),v40,z0,tPen\WObj:=wPaper;
    MoveL Offs(pOrigin,125.60,117.07,0.00),v40,z0,tPen\WObj:=wPaper;
    MoveL Offs(pOrigin,125.75,118.43,0.00),v40,z0,tPen\WObj:=wPaper;
    MoveL Offs(pOrigin,126.50,119.93,0.00),v40,z0,tPen\WObj:=wPaper;
    MoveL Offs(pOrigin,126.50,119.93,0.00),v40,z0,tPen\WObj:=wPaper;
    MoveL Offs(pOrigin,126.10,122.78,0.00),v40,z0,tPen\WObj:=wPaper;
    MoveL Offs(pOrigin,123.95,124.97,0.00),v40,z0,tPen\WObj:=wPaper;
    MoveL Offs(pOrigin,115.25,124.97,0.00),v40,z0,tPen\WObj:=wPaper;
    MoveL Offs(pOrigin,113.45,123.22,0.00),v40,z0,tPen\WObj:=wPaper;
    MoveL Offs(pOrigin,113.20,122.47,0.00),v40,z0,tPen\WObj:=wPaper;
    MoveL Offs(pOrigin,119.75,115.57,0.00),v40,fine,tPen\WObj:=wPaper;
    MoveL Offs(pOrigin,119.75,115.57,6.00),v60,z5,tPen\WObj:=wPaper;
    MoveL Offs(pOrigin,121.10,114.68,6.00),vTravel,z5,tPen\WObj:=wPaper;
    MoveL Offs(pOrigin,121.10,114.68,0.00),v60,z0,tPen\WObj:=wPaper;
    MoveL Offs(pOrigin,119.75,113.93,0.00),v40,z0,tPen\WObj:=wPaper;
    MoveL Offs(pOrigin,119.75,113.93,0.00),v40,z0,tPen\WObj:=wPaper;
    MoveL Offs(pOrigin,112.85,120.53,0.00),v40,fine,tPen\WObj:=wPaper;
    MoveL Offs(pOrigin,112.85,120.53,6.00),v60,z5,tPen\WObj:=wPaper;
    MoveL Offs(pOrigin,113.15,122.32,6.00),vTravel,z5,tPen\WObj:=wPaper;
    MoveL Offs(pOrigin,113.15,122.32,0.00),v60,z0,tPen\WObj:=wPaper;
    MoveL Offs(pOrigin,112.40,120.07,0.00),v40,z0,tPen\WObj:=wPaper;
    MoveL Offs(pOrigin,112.40,118.12,0.00),v40,z0,tPen\WObj:=wPaper;
    MoveL Offs(pOrigin,111.65,115.43,0.00),v40,z0,tPen\WObj:=wPaper;
    MoveL Offs(pOrigin,111.65,106.12,0.00),v40,z0,tPen\WObj:=wPaper;
    MoveL Offs(pOrigin,113.45,104.32,0.00),v40,z0,tPen\WObj:=wPaper;
    MoveL Offs(pOrigin,113.45,104.32,0.00),v40,z0,tPen\WObj:=wPaper;
    MoveL Offs(pOrigin,116.45,107.32,0.00),v40,fine,tPen\WObj:=wPaper;
    MoveL Offs(pOrigin,116.45,107.32,6.00),v60,z5,tPen\WObj:=wPaper;
    MoveL Offs(pOrigin,116.75,113.78,6.00),vTravel,z5,tPen\WObj:=wPaper;
    MoveL Offs(pOrigin,116.75,113.78,0.00),v60,z0,tPen\WObj:=wPaper;
    MoveL Offs(pOrigin,112.40,117.82,0.00),v40,fine,tPen\WObj:=wPaper;
    MoveL Offs(pOrigin,112.40,117.82,6.00),v60,z5,tPen\WObj:=wPaper;
    MoveL Offs(pOrigin,113.45,123.38,6.00),vTravel,z5,tPen\WObj:=wPaper;
    MoveL Offs(pOrigin,113.45,123.38,0.00),v60,z0,tPen\WObj:=wPaper;
    MoveL Offs(pOrigin,114.95,124.88,0.00),v40,z0,tPen\WObj:=wPaper;
    MoveL Offs(pOrigin,113.45,123.38,0.00),v40,fine,tPen\WObj:=wPaper;
    MoveL Offs(pOrigin,113.45,123.38,6.00),v60,z5,tPen\WObj:=wPaper;
    MoveL Offs(pOrigin,119.75,113.93,6.00),vTravel,z5,tPen\WObj:=wPaper;
    MoveL Offs(pOrigin,119.75,113.93,0.00),v60,z0,tPen\WObj:=wPaper;
    MoveL Offs(pOrigin,119.90,113.03,0.00),v40,z0,tPen\WObj:=wPaper;
    MoveL Offs(pOrigin,121.70,111.22,0.00),v40,z0,tPen\WObj:=wPaper;
    MoveL Offs(pOrigin,121.70,111.22,0.00),v40,z0,tPen\WObj:=wPaper;
    MoveL Offs(pOrigin,121.15,110.62,0.00),v40,z0,tPen\WObj:=wPaper;
    MoveL Offs(pOrigin,121.25,110.18,0.00),v40,z0,tPen\WObj:=wPaper;
    MoveL Offs(pOrigin,128.45,102.82,0.00),v40,fine,tPen\WObj:=wPaper;
    MoveL Offs(pOrigin,128.45,102.82,6.00),v60,z5,tPen\WObj:=wPaper;
    MoveL Offs(pOrigin,128.15,101.32,6.00),vTravel,z5,tPen\WObj:=wPaper;
    MoveL Offs(pOrigin,128.15,101.32,0.00),v60,z0,tPen\WObj:=wPaper;
    MoveL Offs(pOrigin,127.25,100.72,0.00),v40,fine,tPen\WObj:=wPaper;
    MoveL Offs(pOrigin,127.25,100.72,6.00),v60,z5,tPen\WObj:=wPaper;
    MoveL Offs(pOrigin,126.50,99.07,6.00),vTravel,z5,tPen\WObj:=wPaper;
    MoveL Offs(pOrigin,126.50,99.07,0.00),v60,z0,tPen\WObj:=wPaper;
    MoveL Offs(pOrigin,130.70,95.18,0.00),v40,z0,tPen\WObj:=wPaper;
    MoveL Offs(pOrigin,130.70,94.88,0.00),v40,z0,tPen\WObj:=wPaper;
    MoveL Offs(pOrigin,129.95,94.28,0.00),v40,z0,tPen\WObj:=wPaper;
    MoveL Offs(pOrigin,130.40,93.82,0.00),v40,fine,tPen\WObj:=wPaper;
    MoveL Offs(pOrigin,130.40,93.82,6.00),v60,z5,tPen\WObj:=wPaper;
    MoveL Offs(pOrigin,128.75,93.53,6.00),vTravel,z5,tPen\WObj:=wPaper;
    MoveL Offs(pOrigin,128.75,93.53,0.00),v60,z0,tPen\WObj:=wPaper;
    MoveL Offs(pOrigin,128.15,93.22,0.00),v40,z0,tPen\WObj:=wPaper;
    MoveL Offs(pOrigin,127.70,93.38,0.00),v40,z0,tPen\WObj:=wPaper;
    MoveL Offs(pOrigin,124.55,96.38,0.00),v40,z0,tPen\WObj:=wPaper;
    MoveL Offs(pOrigin,124.55,96.38,0.00),v40,z0,tPen\WObj:=wPaper;
    MoveL Offs(pOrigin,123.35,95.18,0.00),v40,z0,tPen\WObj:=wPaper;
    MoveL Offs(pOrigin,122.30,95.03,0.00),v40,z0,tPen\WObj:=wPaper;
    MoveL Offs(pOrigin,119.00,94.88,0.00),v40,z0,tPen\WObj:=wPaper;
    MoveL Offs(pOrigin,118.70,95.18,0.00),v40,z0,tPen\WObj:=wPaper;
    MoveL Offs(pOrigin,117.95,95.32,0.00),v40,z0,tPen\WObj:=wPaper;
  ENDPROC

  PROC DrawPart6()
    MoveL Offs(pOrigin,113.60,99.38,0.00),v40,z0,tPen\WObj:=wPaper;
    MoveL Offs(pOrigin,113.45,100.43,0.00),v40,fine,tPen\WObj:=wPaper;
    MoveL Offs(pOrigin,113.45,100.43,6.00),v60,z5,tPen\WObj:=wPaper;
    MoveL Offs(pOrigin,121.70,95.93,6.00),vTravel,z5,tPen\WObj:=wPaper;
    MoveL Offs(pOrigin,121.70,95.93,0.00),v60,z0,tPen\WObj:=wPaper;
    MoveL Offs(pOrigin,122.30,95.03,0.00),v40,z0,tPen\WObj:=wPaper;
    MoveL Offs(pOrigin,122.30,95.03,0.00),v40,z0,tPen\WObj:=wPaper;
    MoveL Offs(pOrigin,123.20,95.18,0.00),v40,z0,tPen\WObj:=wPaper;
    MoveL Offs(pOrigin,125.15,97.57,0.00),v40,fine,tPen\WObj:=wPaper;
    MoveL Offs(pOrigin,125.15,97.57,6.00),v60,z5,tPen\WObj:=wPaper;
    MoveL Offs(pOrigin,126.20,89.93,6.00),vTravel,z5,tPen\WObj:=wPaper;
    MoveL Offs(pOrigin,126.20,89.93,0.00),v60,z0,tPen\WObj:=wPaper;
    MoveL Offs(pOrigin,125.45,89.18,0.00),v40,z0,tPen\WObj:=wPaper;
    MoveL Offs(pOrigin,125.45,89.18,0.00),v40,z0,tPen\WObj:=wPaper;
    MoveL Offs(pOrigin,124.85,89.22,0.00),v40,z0,tPen\WObj:=wPaper;
    MoveL Offs(pOrigin,124.40,89.82,0.00),v40,z0,tPen\WObj:=wPaper;
    MoveL Offs(pOrigin,123.50,89.93,0.00),v40,z0,tPen\WObj:=wPaper;
    MoveL Offs(pOrigin,122.00,89.07,0.00),v40,z0,tPen\WObj:=wPaper;
    MoveL Offs(pOrigin,120.50,88.82,0.00),v40,z0,tPen\WObj:=wPaper;
    MoveL Offs(pOrigin,119.30,87.82,0.00),v40,z0,tPen\WObj:=wPaper;
    MoveL Offs(pOrigin,119.30,87.82,0.00),v40,z0,tPen\WObj:=wPaper;
    MoveL Offs(pOrigin,120.80,86.32,0.00),v40,z0,tPen\WObj:=wPaper;
    MoveL Offs(pOrigin,121.10,85.47,0.00),v40,z0,tPen\WObj:=wPaper;
    MoveL Offs(pOrigin,122.45,85.12,0.00),v40,z0,tPen\WObj:=wPaper;
    MoveL Offs(pOrigin,126.20,81.38,0.00),v40,z0,tPen\WObj:=wPaper;
    MoveL Offs(pOrigin,125.75,80.47,0.00),v40,z0,tPen\WObj:=wPaper;
    MoveL Offs(pOrigin,122.30,81.53,0.00),v40,z0,tPen\WObj:=wPaper;
    MoveL Offs(pOrigin,118.70,81.53,0.00),v40,z0,tPen\WObj:=wPaper;
    MoveL Offs(pOrigin,117.80,81.97,0.00),v40,z0,tPen\WObj:=wPaper;
    MoveL Offs(pOrigin,117.80,81.97,0.00),v40,z0,tPen\WObj:=wPaper;
    MoveL Offs(pOrigin,120.65,84.68,0.00),v40,z0,tPen\WObj:=wPaper;
    MoveL Offs(pOrigin,120.95,85.43,0.00),v40,fine,tPen\WObj:=wPaper;
    MoveL Offs(pOrigin,120.95,85.43,6.00),v60,z5,tPen\WObj:=wPaper;
    MoveL Offs(pOrigin,121.55,86.62,6.00),vTravel,z5,tPen\WObj:=wPaper;
    MoveL Offs(pOrigin,121.55,86.62,0.00),v60,z0,tPen\WObj:=wPaper;
    MoveL Offs(pOrigin,119.90,88.12,0.00),v40,z0,tPen\WObj:=wPaper;
    MoveL Offs(pOrigin,119.30,87.82,0.00),v40,z0,tPen\WObj:=wPaper;
    MoveL Offs(pOrigin,117.35,87.78,0.00),v40,z0,tPen\WObj:=wPaper;
    MoveL Offs(pOrigin,114.50,84.97,0.00),v40,z0,tPen\WObj:=wPaper;
    MoveL Offs(pOrigin,114.50,84.97,0.00),v40,z0,tPen\WObj:=wPaper;
    MoveL Offs(pOrigin,117.20,82.12,0.00),v40,z0,tPen\WObj:=wPaper;
    MoveL Offs(pOrigin,117.80,81.97,0.00),v40,z0,tPen\WObj:=wPaper;
    MoveL Offs(pOrigin,117.80,81.97,0.00),v40,z0,tPen\WObj:=wPaper;
    MoveL Offs(pOrigin,120.05,84.38,0.00),v40,fine,tPen\WObj:=wPaper;
    MoveL Offs(pOrigin,120.05,84.38,6.00),v60,z5,tPen\WObj:=wPaper;
    MoveL Offs(pOrigin,121.85,86.62,6.00),vTravel,z5,tPen\WObj:=wPaper;
    MoveL Offs(pOrigin,121.85,86.62,0.00),v60,z0,tPen\WObj:=wPaper;
    MoveL Offs(pOrigin,122.15,86.78,0.00),v40,z0,tPen\WObj:=wPaper;
    MoveL Offs(pOrigin,123.35,86.03,0.00),v40,z0,tPen\WObj:=wPaper;
    MoveL Offs(pOrigin,123.35,86.03,0.00),v40,z0,tPen\WObj:=wPaper;
    MoveL Offs(pOrigin,123.35,86.93,0.00),v40,z0,tPen\WObj:=wPaper;
    MoveL Offs(pOrigin,123.35,86.93,0.00),v40,z0,tPen\WObj:=wPaper;
    MoveL Offs(pOrigin,121.70,88.88,0.00),v40,z0,tPen\WObj:=wPaper;
    MoveL Offs(pOrigin,122.15,89.03,0.00),v40,z0,tPen\WObj:=wPaper;
    MoveL Offs(pOrigin,123.95,87.38,0.00),v40,z0,tPen\WObj:=wPaper;
    MoveL Offs(pOrigin,123.80,87.07,0.00),v40,z0,tPen\WObj:=wPaper;
    MoveL Offs(pOrigin,128.00,82.88,0.00),v40,z0,tPen\WObj:=wPaper;
    MoveL Offs(pOrigin,127.10,82.12,0.00),v40,z0,tPen\WObj:=wPaper;
    MoveL Offs(pOrigin,128.25,83.03,0.00),v40,z0,tPen\WObj:=wPaper;
    MoveL Offs(pOrigin,128.30,83.93,0.00),v40,z0,tPen\WObj:=wPaper;
    MoveL Offs(pOrigin,129.35,86.47,0.00),v40,z0,tPen\WObj:=wPaper;
    MoveL Offs(pOrigin,129.35,87.53,0.00),v40,z0,tPen\WObj:=wPaper;
    MoveL Offs(pOrigin,127.25,89.62,0.00),v40,z0,tPen\WObj:=wPaper;
    MoveL Offs(pOrigin,126.20,89.93,0.00),v40,z0,tPen\WObj:=wPaper;
    MoveL Offs(pOrigin,125.45,89.18,0.00),v40,z0,tPen\WObj:=wPaper;
    MoveL Offs(pOrigin,125.60,88.72,0.00),v40,z0,tPen\WObj:=wPaper;
    MoveL Offs(pOrigin,126.05,88.88,0.00),v40,z0,tPen\WObj:=wPaper;
    MoveL Offs(pOrigin,126.20,88.57,0.00),v40,z0,tPen\WObj:=wPaper;
    MoveL Offs(pOrigin,126.20,88.57,0.00),v40,z0,tPen\WObj:=wPaper;
    MoveL Offs(pOrigin,128.90,85.72,0.00),v40,fine,tPen\WObj:=wPaper;
    MoveL Offs(pOrigin,128.90,85.72,6.00),v60,z5,tPen\WObj:=wPaper;
    MoveL Offs(pOrigin,128.30,84.22,6.00),vTravel,z5,tPen\WObj:=wPaper;
    MoveL Offs(pOrigin,128.30,84.22,0.00),v60,z0,tPen\WObj:=wPaper;
    MoveL Offs(pOrigin,124.45,87.82,0.00),v40,z0,tPen\WObj:=wPaper;
    MoveL Offs(pOrigin,124.35,88.72,0.00),v40,z0,tPen\WObj:=wPaper;
    MoveL Offs(pOrigin,124.70,89.18,0.00),v40,z0,tPen\WObj:=wPaper;
    MoveL Offs(pOrigin,124.25,88.88,0.00),v40,z0,tPen\WObj:=wPaper;
    MoveL Offs(pOrigin,123.50,88.88,0.00),v40,z0,tPen\WObj:=wPaper;
    MoveL Offs(pOrigin,123.05,89.47,0.00),v40,fine,tPen\WObj:=wPaper;
    MoveL Offs(pOrigin,123.05,89.47,6.00),v60,z5,tPen\WObj:=wPaper;
    MoveL Offs(pOrigin,123.35,86.03,6.00),vTravel,z5,tPen\WObj:=wPaper;
    MoveL Offs(pOrigin,123.35,86.03,0.00),v60,z0,tPen\WObj:=wPaper;
    MoveL Offs(pOrigin,127.10,82.12,0.00),v40,fine,tPen\WObj:=wPaper;
    MoveL Offs(pOrigin,127.10,82.12,6.00),v60,z5,tPen\WObj:=wPaper;
    MoveL Offs(pOrigin,125.60,79.43,6.00),vTravel,z5,tPen\WObj:=wPaper;
    MoveL Offs(pOrigin,125.60,79.43,0.00),v60,z0,tPen\WObj:=wPaper;
    MoveL Offs(pOrigin,123.30,74.32,0.00),v40,z0,tPen\WObj:=wPaper;
    MoveL Offs(pOrigin,121.70,73.72,0.00),v40,z0,tPen\WObj:=wPaper;
    MoveL Offs(pOrigin,121.70,73.72,0.00),v40,z0,tPen\WObj:=wPaper;
    MoveL Offs(pOrigin,120.80,73.12,0.00),v40,z0,tPen\WObj:=wPaper;
    MoveL Offs(pOrigin,118.50,75.47,0.00),v40,z0,tPen\WObj:=wPaper;
    MoveL Offs(pOrigin,116.75,76.28,0.00),v40,z0,tPen\WObj:=wPaper;
    MoveL Offs(pOrigin,116.75,76.28,0.00),v40,z0,tPen\WObj:=wPaper;
    MoveL Offs(pOrigin,112.40,80.47,0.00),v40,z0,tPen\WObj:=wPaper;
    MoveL Offs(pOrigin,112.40,80.47,0.00),v40,z0,tPen\WObj:=wPaper;
    MoveL Offs(pOrigin,112.40,82.43,0.00),v40,z0,tPen\WObj:=wPaper;
    MoveL Offs(pOrigin,112.85,83.03,0.00),v40,z0,tPen\WObj:=wPaper;
    MoveL Offs(pOrigin,112.85,83.03,0.00),v40,z0,tPen\WObj:=wPaper;
    MoveL Offs(pOrigin,112.90,84.53,0.00),v40,z0,tPen\WObj:=wPaper;
    MoveL Offs(pOrigin,114.50,85.12,0.00),v40,z0,tPen\WObj:=wPaper;
    MoveL Offs(pOrigin,117.20,87.82,0.00),v40,fine,tPen\WObj:=wPaper;
    MoveL Offs(pOrigin,117.20,87.82,6.00),v60,z5,tPen\WObj:=wPaper;
    MoveL Offs(pOrigin,112.85,83.03,6.00),vTravel,z5,tPen\WObj:=wPaper;
    MoveL Offs(pOrigin,112.85,83.03,0.00),v60,z0,tPen\WObj:=wPaper;
    MoveL Offs(pOrigin,119.75,76.43,0.00),v40,z0,tPen\WObj:=wPaper;
    MoveL Offs(pOrigin,119.75,76.43,0.00),v40,z0,tPen\WObj:=wPaper;
    MoveL Offs(pOrigin,120.65,76.72,0.00),v40,z0,tPen\WObj:=wPaper;
    MoveL Offs(pOrigin,120.95,77.18,0.00),v40,fine,tPen\WObj:=wPaper;
    MoveL Offs(pOrigin,120.95,77.18,6.00),v60,z5,tPen\WObj:=wPaper;
    MoveL Offs(pOrigin,119.75,76.43,6.00),vTravel,z5,tPen\WObj:=wPaper;
    MoveL Offs(pOrigin,119.75,76.43,0.00),v60,z0,tPen\WObj:=wPaper;
    MoveL Offs(pOrigin,119.90,75.53,0.00),v40,z0,tPen\WObj:=wPaper;
    MoveL Offs(pOrigin,121.70,73.72,0.00),v40,z0,tPen\WObj:=wPaper;
    MoveL Offs(pOrigin,121.70,73.72,0.00),v40,z0,tPen\WObj:=wPaper;
    MoveL Offs(pOrigin,121.10,72.97,0.00),v40,z0,tPen\WObj:=wPaper;
    MoveL Offs(pOrigin,119.90,72.38,0.00),v40,z0,tPen\WObj:=wPaper;
    MoveL Offs(pOrigin,119.90,72.38,0.00),v40,z0,tPen\WObj:=wPaper;
    MoveL Offs(pOrigin,119.60,71.47,0.00),v40,z0,tPen\WObj:=wPaper;
    MoveL Offs(pOrigin,119.60,71.47,0.00),v40,z0,tPen\WObj:=wPaper;
    MoveL Offs(pOrigin,121.40,69.53,0.00),v40,z0,tPen\WObj:=wPaper;
  ENDPROC

  PROC DrawPart7()
    MoveL Offs(pOrigin,122.30,67.72,0.00),v40,z0,tPen\WObj:=wPaper;
    MoveL Offs(pOrigin,122.60,67.57,0.00),v40,z0,tPen\WObj:=wPaper;
    MoveL Offs(pOrigin,127.55,62.92,0.00),v40,z0,tPen\WObj:=wPaper;
    MoveL Offs(pOrigin,127.55,62.92,0.00),v40,z0,tPen\WObj:=wPaper;
    MoveL Offs(pOrigin,128.10,63.53,0.00),v40,z0,tPen\WObj:=wPaper;
    MoveL Offs(pOrigin,128.45,65.47,0.00),v40,z0,tPen\WObj:=wPaper;
    MoveL Offs(pOrigin,128.45,65.47,0.00),v40,z0,tPen\WObj:=wPaper;
    MoveL Offs(pOrigin,128.90,65.78,0.00),v40,z0,tPen\WObj:=wPaper;
    MoveL Offs(pOrigin,129.05,66.53,0.00),v40,z0,tPen\WObj:=wPaper;
    MoveL Offs(pOrigin,129.05,66.53,0.00),v40,z0,tPen\WObj:=wPaper;
    MoveL Offs(pOrigin,129.50,66.97,0.00),v40,z0,tPen\WObj:=wPaper;
    MoveL Offs(pOrigin,129.50,68.18,0.00),v40,z0,tPen\WObj:=wPaper;
    MoveL Offs(pOrigin,129.50,68.18,0.00),v40,z0,tPen\WObj:=wPaper;
    MoveL Offs(pOrigin,129.80,68.47,0.00),v40,z0,tPen\WObj:=wPaper;
    MoveL Offs(pOrigin,129.80,69.82,0.00),v40,z0,tPen\WObj:=wPaper;
    MoveL Offs(pOrigin,129.80,69.82,0.00),v40,z0,tPen\WObj:=wPaper;
    MoveL Offs(pOrigin,131.05,71.18,0.00),v40,z0,tPen\WObj:=wPaper;
    MoveL Offs(pOrigin,131.15,73.12,0.00),v40,z0,tPen\WObj:=wPaper;
    MoveL Offs(pOrigin,131.15,73.12,0.00),v40,z0,tPen\WObj:=wPaper;
    MoveL Offs(pOrigin,131.60,74.18,0.00),v40,z0,tPen\WObj:=wPaper;
    MoveL Offs(pOrigin,131.60,75.53,0.00),v40,z0,tPen\WObj:=wPaper;
    MoveL Offs(pOrigin,130.55,76.57,0.00),v40,fine,tPen\WObj:=wPaper;
    MoveL Offs(pOrigin,130.55,76.57,6.00),v60,z5,tPen\WObj:=wPaper;
    MoveL Offs(pOrigin,131.00,70.88,6.00),vTravel,z5,tPen\WObj:=wPaper;
    MoveL Offs(pOrigin,131.00,70.88,0.00),v60,z0,tPen\WObj:=wPaper;
    MoveL Offs(pOrigin,129.80,69.82,0.00),v40,z0,tPen\WObj:=wPaper;
    MoveL Offs(pOrigin,129.80,69.82,0.00),v40,z0,tPen\WObj:=wPaper;
    MoveL Offs(pOrigin,129.05,70.57,0.00),v40,z0,tPen\WObj:=wPaper;
    MoveL Offs(pOrigin,129.05,70.57,0.00),v40,z0,tPen\WObj:=wPaper;
    MoveL Offs(pOrigin,128.85,72.53,0.00),v40,z0,tPen\WObj:=wPaper;
    MoveL Offs(pOrigin,124.55,76.43,0.00),v40,fine,tPen\WObj:=wPaper;
    MoveL Offs(pOrigin,124.55,76.43,6.00),v60,z5,tPen\WObj:=wPaper;
    MoveL Offs(pOrigin,121.10,72.82,6.00),vTravel,z5,tPen\WObj:=wPaper;
    MoveL Offs(pOrigin,121.10,72.82,0.00),v60,z0,tPen\WObj:=wPaper;
    MoveL Offs(pOrigin,128.45,65.47,0.00),v40,fine,tPen\WObj:=wPaper;
    MoveL Offs(pOrigin,128.45,65.47,6.00),v60,z5,tPen\WObj:=wPaper;
    MoveL Offs(pOrigin,129.05,66.53,6.00),vTravel,z5,tPen\WObj:=wPaper;
    MoveL Offs(pOrigin,129.05,66.53,0.00),v60,z0,tPen\WObj:=wPaper;
    MoveL Offs(pOrigin,126.65,68.93,0.00),v40,z0,tPen\WObj:=wPaper;
    MoveL Offs(pOrigin,126.55,69.68,0.00),v40,z0,tPen\WObj:=wPaper;
    MoveL Offs(pOrigin,127.70,69.78,0.00),v40,z0,tPen\WObj:=wPaper;
    MoveL Offs(pOrigin,129.50,68.18,0.00),v40,fine,tPen\WObj:=wPaper;
    MoveL Offs(pOrigin,129.50,68.18,6.00),v60,z5,tPen\WObj:=wPaper;
    MoveL Offs(pOrigin,127.55,62.92,6.00),vTravel,z5,tPen\WObj:=wPaper;
    MoveL Offs(pOrigin,127.55,62.92,0.00),v60,z0,tPen\WObj:=wPaper;
    MoveL Offs(pOrigin,127.55,62.03,0.00),v40,z0,tPen\WObj:=wPaper;
    MoveL Offs(pOrigin,127.10,61.58,0.00),v40,z0,tPen\WObj:=wPaper;
    MoveL Offs(pOrigin,127.10,61.58,0.00),v40,z0,tPen\WObj:=wPaper;
    MoveL Offs(pOrigin,127.10,60.38,0.00),v40,z0,tPen\WObj:=wPaper;
    MoveL Offs(pOrigin,126.80,60.08,0.00),v40,z0,tPen\WObj:=wPaper;
    MoveL Offs(pOrigin,126.80,60.08,0.00),v40,z0,tPen\WObj:=wPaper;
    MoveL Offs(pOrigin,126.65,59.47,0.00),v40,z0,tPen\WObj:=wPaper;
    MoveL Offs(pOrigin,124.70,57.83,0.00),v40,z0,tPen\WObj:=wPaper;
    MoveL Offs(pOrigin,114.35,57.83,0.00),v40,z0,tPen\WObj:=wPaper;
    MoveL Offs(pOrigin,113.85,58.28,0.00),v40,z0,tPen\WObj:=wPaper;
    MoveL Offs(pOrigin,113.60,59.17,0.00),v40,z0,tPen\WObj:=wPaper;
    MoveL Offs(pOrigin,113.60,59.17,0.00),v40,z0,tPen\WObj:=wPaper;
    MoveL Offs(pOrigin,120.35,65.78,0.00),v40,z0,tPen\WObj:=wPaper;
    MoveL Offs(pOrigin,120.05,65.47,0.00),v40,z0,tPen\WObj:=wPaper;
    MoveL Offs(pOrigin,113.60,59.17,0.00),v40,z0,tPen\WObj:=wPaper;
    MoveL Offs(pOrigin,113.60,59.17,0.00),v40,z0,tPen\WObj:=wPaper;
    MoveL Offs(pOrigin,113.45,66.22,0.00),v40,z0,tPen\WObj:=wPaper;
    MoveL Offs(pOrigin,113.45,66.22,0.00),v40,z0,tPen\WObj:=wPaper;
    MoveL Offs(pOrigin,116.60,69.38,0.00),v40,z0,tPen\WObj:=wPaper;
    MoveL Offs(pOrigin,117.95,69.97,0.00),v40,z0,tPen\WObj:=wPaper;
    MoveL Offs(pOrigin,119.30,71.47,0.00),v40,z0,tPen\WObj:=wPaper;
    MoveL Offs(pOrigin,119.30,71.47,0.00),v40,z0,tPen\WObj:=wPaper;
    MoveL Offs(pOrigin,117.50,73.22,0.00),v40,z0,tPen\WObj:=wPaper;
    MoveL Offs(pOrigin,116.75,72.97,0.00),v40,z0,tPen\WObj:=wPaper;
    MoveL Offs(pOrigin,116.90,73.28,0.00),v40,z0,tPen\WObj:=wPaper;
    MoveL Offs(pOrigin,111.80,68.47,0.00),v40,z0,tPen\WObj:=wPaper;
    MoveL Offs(pOrigin,111.80,68.47,0.00),v40,z0,tPen\WObj:=wPaper;
    MoveL Offs(pOrigin,111.95,67.57,0.00),v40,z0,tPen\WObj:=wPaper;
    MoveL Offs(pOrigin,113.45,66.22,0.00),v40,z0,tPen\WObj:=wPaper;
    MoveL Offs(pOrigin,113.45,66.22,0.00),v40,z0,tPen\WObj:=wPaper;
    MoveL Offs(pOrigin,116.75,69.38,0.00),v40,fine,tPen\WObj:=wPaper;
    MoveL Offs(pOrigin,116.75,69.38,6.00),v60,z5,tPen\WObj:=wPaper;
    MoveL Offs(pOrigin,117.95,69.82,6.00),vTravel,z5,tPen\WObj:=wPaper;
    MoveL Offs(pOrigin,117.95,69.82,0.00),v60,z0,tPen\WObj:=wPaper;
    MoveL Offs(pOrigin,119.60,68.03,0.00),v40,z0,tPen\WObj:=wPaper;
    MoveL Offs(pOrigin,121.40,67.38,0.00),v40,z0,tPen\WObj:=wPaper;
    MoveL Offs(pOrigin,121.55,66.82,0.00),v40,z0,tPen\WObj:=wPaper;
    MoveL Offs(pOrigin,121.55,66.82,0.00),v40,z0,tPen\WObj:=wPaper;
    MoveL Offs(pOrigin,122.30,66.53,0.00),v40,z0,tPen\WObj:=wPaper;
    MoveL Offs(pOrigin,127.10,61.58,0.00),v40,fine,tPen\WObj:=wPaper;
    MoveL Offs(pOrigin,127.10,61.58,6.00),v60,z5,tPen\WObj:=wPaper;
    MoveL Offs(pOrigin,126.80,60.08,6.00),vTravel,z5,tPen\WObj:=wPaper;
    MoveL Offs(pOrigin,126.80,60.08,0.00),v60,z0,tPen\WObj:=wPaper;
    MoveL Offs(pOrigin,121.25,65.62,0.00),v40,z0,tPen\WObj:=wPaper;
    MoveL Offs(pOrigin,121.10,66.22,0.00),v40,fine,tPen\WObj:=wPaper;
    MoveL Offs(pOrigin,121.10,66.22,6.00),v60,z5,tPen\WObj:=wPaper;
    MoveL Offs(pOrigin,118.85,70.88,6.00),vTravel,z5,tPen\WObj:=wPaper;
    MoveL Offs(pOrigin,118.85,70.88,0.00),v60,z0,tPen\WObj:=wPaper;
    MoveL Offs(pOrigin,119.60,71.47,0.00),v40,z0,tPen\WObj:=wPaper;
    MoveL Offs(pOrigin,119.90,72.38,0.00),v40,z0,tPen\WObj:=wPaper;
    MoveL Offs(pOrigin,117.65,74.62,0.00),v40,z0,tPen\WObj:=wPaper;
    MoveL Offs(pOrigin,117.45,75.68,0.00),v40,z0,tPen\WObj:=wPaper;
    MoveL Offs(pOrigin,116.90,75.97,0.00),v40,z0,tPen\WObj:=wPaper;
    MoveL Offs(pOrigin,116.75,75.38,0.00),v40,z0,tPen\WObj:=wPaper;
    MoveL Offs(pOrigin,116.60,75.07,0.00),v40,z0,tPen\WObj:=wPaper;
    MoveL Offs(pOrigin,116.45,75.38,0.00),v40,z0,tPen\WObj:=wPaper;
    MoveL Offs(pOrigin,116.75,75.38,0.00),v40,z0,tPen\WObj:=wPaper;
    MoveL Offs(pOrigin,116.45,75.07,0.00),v40,z0,tPen\WObj:=wPaper;
    MoveL Offs(pOrigin,116.45,75.38,0.00),v40,z0,tPen\WObj:=wPaper;
    MoveL Offs(pOrigin,116.75,75.38,0.00),v40,z0,tPen\WObj:=wPaper;
    MoveL Offs(pOrigin,116.45,75.38,0.00),v40,z0,tPen\WObj:=wPaper;
    MoveL Offs(pOrigin,112.10,79.43,0.00),v40,z0,tPen\WObj:=wPaper;
    MoveL Offs(pOrigin,112.40,80.47,0.00),v40,z0,tPen\WObj:=wPaper;
    MoveL Offs(pOrigin,111.50,77.62,0.00),v40,z0,tPen\WObj:=wPaper;
    MoveL Offs(pOrigin,111.50,68.78,0.00),v40,z0,tPen\WObj:=wPaper;
    MoveL Offs(pOrigin,111.80,68.47,0.00),v40,z0,tPen\WObj:=wPaper;
    MoveL Offs(pOrigin,111.80,68.47,0.00),v40,z0,tPen\WObj:=wPaper;
    MoveL Offs(pOrigin,116.15,72.68,0.00),v40,z0,tPen\WObj:=wPaper;
    MoveL Offs(pOrigin,116.90,73.28,0.00),v40,z0,tPen\WObj:=wPaper;
    MoveL Offs(pOrigin,116.60,73.88,0.00),v40,z0,tPen\WObj:=wPaper;
    MoveL Offs(pOrigin,111.95,78.22,0.00),v40,fine,tPen\WObj:=wPaper;
    MoveL Offs(pOrigin,111.95,78.22,6.00),v60,z5,tPen\WObj:=wPaper;
    MoveL Offs(pOrigin,125.60,58.58,6.00),vTravel,z5,tPen\WObj:=wPaper;
    MoveL Offs(pOrigin,125.60,58.58,0.00),v60,z0,tPen\WObj:=wPaper;
    MoveL Offs(pOrigin,126.65,59.62,0.00),v40,z0,tPen\WObj:=wPaper;
  ENDPROC

  PROC DrawPart8()
    MoveL Offs(pOrigin,125.60,58.58,0.00),v40,fine,tPen\WObj:=wPaper;
    MoveL Offs(pOrigin,125.60,58.58,6.00),v60,z5,tPen\WObj:=wPaper;
    MoveL Offs(pOrigin,135.05,69.68,6.00),vTravel,z5,tPen\WObj:=wPaper;
    MoveL Offs(pOrigin,135.05,69.68,0.00),v60,z0,tPen\WObj:=wPaper;
    MoveL Offs(pOrigin,134.90,69.82,0.00),v40,z0,tPen\WObj:=wPaper;
    MoveL Offs(pOrigin,135.95,70.57,0.00),v40,z0,tPen\WObj:=wPaper;
    MoveL Offs(pOrigin,135.95,70.57,0.00),v40,z0,tPen\WObj:=wPaper;
    MoveL Offs(pOrigin,137.15,69.97,0.00),v40,z0,tPen\WObj:=wPaper;
    MoveL Offs(pOrigin,137.15,69.97,0.00),v40,z0,tPen\WObj:=wPaper;
    MoveL Offs(pOrigin,138.05,68.47,0.00),v40,z0,tPen\WObj:=wPaper;
    MoveL Offs(pOrigin,141.65,65.03,0.00),v40,fine,tPen\WObj:=wPaper;
    MoveL Offs(pOrigin,141.65,65.03,6.00),v60,z5,tPen\WObj:=wPaper;
    MoveL Offs(pOrigin,140.75,62.62,6.00),vTravel,z5,tPen\WObj:=wPaper;
    MoveL Offs(pOrigin,140.75,62.62,0.00),v60,z0,tPen\WObj:=wPaper;
    MoveL Offs(pOrigin,140.75,61.88,0.00),v40,z0,tPen\WObj:=wPaper;
    MoveL Offs(pOrigin,140.30,61.42,0.00),v40,z0,tPen\WObj:=wPaper;
    MoveL Offs(pOrigin,140.30,61.42,0.00),v40,z0,tPen\WObj:=wPaper;
    MoveL Offs(pOrigin,140.45,59.78,0.00),v40,z0,tPen\WObj:=wPaper;
    MoveL Offs(pOrigin,140.90,59.33,0.00),v40,z0,tPen\WObj:=wPaper;
    MoveL Offs(pOrigin,140.90,59.33,0.00),v40,z0,tPen\WObj:=wPaper;
    MoveL Offs(pOrigin,146.45,64.88,0.00),v40,z0,tPen\WObj:=wPaper;
    MoveL Offs(pOrigin,147.05,65.78,0.00),v40,z0,tPen\WObj:=wPaper;
    MoveL Offs(pOrigin,147.35,66.68,0.00),v40,z0,tPen\WObj:=wPaper;
    MoveL Offs(pOrigin,147.35,66.68,0.00),v40,z0,tPen\WObj:=wPaper;
    MoveL Offs(pOrigin,147.05,67.53,0.00),v40,z0,tPen\WObj:=wPaper;
    MoveL Offs(pOrigin,145.40,67.93,0.00),v40,z0,tPen\WObj:=wPaper;
    MoveL Offs(pOrigin,143.90,69.38,0.00),v40,z0,tPen\WObj:=wPaper;
    MoveL Offs(pOrigin,143.90,69.38,0.00),v40,z0,tPen\WObj:=wPaper;
    MoveL Offs(pOrigin,144.95,70.53,0.00),v40,z0,tPen\WObj:=wPaper;
    MoveL Offs(pOrigin,146.45,70.57,0.00),v40,z0,tPen\WObj:=wPaper;
    MoveL Offs(pOrigin,146.45,70.57,0.00),v40,z0,tPen\WObj:=wPaper;
    MoveL Offs(pOrigin,147.05,71.47,0.00),v40,z0,tPen\WObj:=wPaper;
    MoveL Offs(pOrigin,147.80,71.62,0.00),v40,fine,tPen\WObj:=wPaper;
    MoveL Offs(pOrigin,147.80,71.62,6.00),v60,z5,tPen\WObj:=wPaper;
    MoveL Offs(pOrigin,146.45,70.57,6.00),vTravel,z5,tPen\WObj:=wPaper;
    MoveL Offs(pOrigin,146.45,70.57,0.00),v60,z0,tPen\WObj:=wPaper;
    MoveL Offs(pOrigin,147.30,69.68,0.00),v40,z0,tPen\WObj:=wPaper;
    MoveL Offs(pOrigin,147.80,68.18,0.00),v40,z0,tPen\WObj:=wPaper;
    MoveL Offs(pOrigin,149.00,67.22,0.00),v40,z0,tPen\WObj:=wPaper;
    MoveL Offs(pOrigin,150.15,69.07,0.00),v40,z0,tPen\WObj:=wPaper;
    MoveL Offs(pOrigin,150.05,69.97,0.00),v40,z0,tPen\WObj:=wPaper;
    MoveL Offs(pOrigin,150.05,69.97,0.00),v40,z0,tPen\WObj:=wPaper;
    MoveL Offs(pOrigin,149.15,70.43,0.00),v40,z0,tPen\WObj:=wPaper;
    MoveL Offs(pOrigin,147.85,71.78,0.00),v40,z0,tPen\WObj:=wPaper;
    MoveL Offs(pOrigin,148.10,73.72,0.00),v40,z0,tPen\WObj:=wPaper;
    MoveL Offs(pOrigin,148.10,73.72,0.00),v40,z0,tPen\WObj:=wPaper;
    MoveL Offs(pOrigin,149.30,74.18,0.00),v40,z0,tPen\WObj:=wPaper;
    MoveL Offs(pOrigin,150.80,77.78,0.00),v40,z0,tPen\WObj:=wPaper;
    MoveL Offs(pOrigin,153.65,80.62,0.00),v40,z0,tPen\WObj:=wPaper;
    MoveL Offs(pOrigin,153.65,80.62,0.00),v40,z0,tPen\WObj:=wPaper;
    MoveL Offs(pOrigin,154.55,80.68,0.00),v40,z0,tPen\WObj:=wPaper;
    MoveL Offs(pOrigin,155.60,81.53,0.00),v40,z0,tPen\WObj:=wPaper;
    MoveL Offs(pOrigin,155.60,81.53,0.00),v40,z0,tPen\WObj:=wPaper;
    MoveL Offs(pOrigin,159.05,79.57,0.00),v40,z0,tPen\WObj:=wPaper;
    MoveL Offs(pOrigin,159.05,75.53,0.00),v40,z0,tPen\WObj:=wPaper;
    MoveL Offs(pOrigin,158.30,70.57,0.00),v40,z0,tPen\WObj:=wPaper;
    MoveL Offs(pOrigin,158.00,70.28,0.00),v40,z0,tPen\WObj:=wPaper;
    MoveL Offs(pOrigin,158.00,70.28,0.00),v40,z0,tPen\WObj:=wPaper;
    MoveL Offs(pOrigin,154.80,73.38,0.00),v40,z0,tPen\WObj:=wPaper;
    MoveL Offs(pOrigin,154.25,73.28,0.00),v40,z0,tPen\WObj:=wPaper;
    MoveL Offs(pOrigin,152.90,74.18,0.00),v40,z0,tPen\WObj:=wPaper;
    MoveL Offs(pOrigin,150.50,76.43,0.00),v40,fine,tPen\WObj:=wPaper;
    MoveL Offs(pOrigin,150.50,76.43,6.00),v60,z5,tPen\WObj:=wPaper;
    MoveL Offs(pOrigin,150.80,77.62,6.00),vTravel,z5,tPen\WObj:=wPaper;
    MoveL Offs(pOrigin,150.80,77.62,0.00),v60,z0,tPen\WObj:=wPaper;
    MoveL Offs(pOrigin,153.65,80.62,0.00),v40,z0,tPen\WObj:=wPaper;
    MoveL Offs(pOrigin,154.70,80.62,0.00),v40,z0,tPen\WObj:=wPaper;
    MoveL Offs(pOrigin,155.60,81.53,0.00),v40,z0,tPen\WObj:=wPaper;
    MoveL Offs(pOrigin,155.60,81.53,0.00),v40,z0,tPen\WObj:=wPaper;
    MoveL Offs(pOrigin,155.00,84.07,0.00),v40,z0,tPen\WObj:=wPaper;
    MoveL Offs(pOrigin,150.50,88.57,0.00),v40,z0,tPen\WObj:=wPaper;
    MoveL Offs(pOrigin,146.60,88.72,0.00),v40,z0,tPen\WObj:=wPaper;
    MoveL Offs(pOrigin,146.15,88.28,0.00),v40,z0,tPen\WObj:=wPaper;
    MoveL Offs(pOrigin,146.15,88.28,0.00),v40,z0,tPen\WObj:=wPaper;
    MoveL Offs(pOrigin,147.05,86.93,0.00),v40,z0,tPen\WObj:=wPaper;
    MoveL Offs(pOrigin,147.35,86.93,0.00),v40,z0,tPen\WObj:=wPaper;
    MoveL Offs(pOrigin,147.80,86.93,0.00),v40,z0,tPen\WObj:=wPaper;
    MoveL Offs(pOrigin,147.95,86.32,0.00),v40,z0,tPen\WObj:=wPaper;
    MoveL Offs(pOrigin,148.10,85.72,0.00),v40,z0,tPen\WObj:=wPaper;
    MoveL Offs(pOrigin,149.00,85.43,0.00),v40,z0,tPen\WObj:=wPaper;
    MoveL Offs(pOrigin,153.35,80.82,0.00),v40,z0,tPen\WObj:=wPaper;
    MoveL Offs(pOrigin,149.75,80.93,0.00),v40,z0,tPen\WObj:=wPaper;
    MoveL Offs(pOrigin,147.50,81.68,0.00),v40,z0,tPen\WObj:=wPaper;
    MoveL Offs(pOrigin,144.50,81.68,0.00),v40,z0,tPen\WObj:=wPaper;
    MoveL Offs(pOrigin,143.00,82.28,0.00),v40,z0,tPen\WObj:=wPaper;
    MoveL Offs(pOrigin,141.50,83.78,0.00),v40,z0,tPen\WObj:=wPaper;
    MoveL Offs(pOrigin,141.50,83.78,0.00),v40,z0,tPen\WObj:=wPaper;
    MoveL Offs(pOrigin,141.05,82.72,0.00),v40,z0,tPen\WObj:=wPaper;
    MoveL Offs(pOrigin,141.05,82.72,0.00),v40,z0,tPen\WObj:=wPaper;
    MoveL Offs(pOrigin,144.00,79.72,0.00),v40,z0,tPen\WObj:=wPaper;
    MoveL Offs(pOrigin,143.90,78.07,0.00),v40,z0,tPen\WObj:=wPaper;
    MoveL Offs(pOrigin,143.90,78.07,0.00),v40,z0,tPen\WObj:=wPaper;
    MoveL Offs(pOrigin,142.85,78.22,0.00),v40,z0,tPen\WObj:=wPaper;
    MoveL Offs(pOrigin,142.85,78.22,0.00),v40,z0,tPen\WObj:=wPaper;
    MoveL Offs(pOrigin,139.55,81.38,0.00),v40,z0,tPen\WObj:=wPaper;
    MoveL Offs(pOrigin,139.55,81.38,0.00),v40,z0,tPen\WObj:=wPaper;
    MoveL Offs(pOrigin,139.85,82.57,0.00),v40,z0,tPen\WObj:=wPaper;
    MoveL Offs(pOrigin,141.05,82.72,0.00),v40,fine,tPen\WObj:=wPaper;
    MoveL Offs(pOrigin,141.05,82.72,6.00),v60,z5,tPen\WObj:=wPaper;
    MoveL Offs(pOrigin,141.50,84.07,6.00),vTravel,z5,tPen\WObj:=wPaper;
    MoveL Offs(pOrigin,141.50,84.07,0.00),v60,z0,tPen\WObj:=wPaper;
    MoveL Offs(pOrigin,141.95,84.53,0.00),v40,z0,tPen\WObj:=wPaper;
    MoveL Offs(pOrigin,141.95,85.43,0.00),v40,z0,tPen\WObj:=wPaper;
    MoveL Offs(pOrigin,141.95,85.43,0.00),v40,z0,tPen\WObj:=wPaper;
    MoveL Offs(pOrigin,142.40,86.03,0.00),v40,z0,tPen\WObj:=wPaper;
    MoveL Offs(pOrigin,142.40,87.22,0.00),v40,z0,tPen\WObj:=wPaper;
    MoveL Offs(pOrigin,142.40,87.22,0.00),v40,z0,tPen\WObj:=wPaper;
    MoveL Offs(pOrigin,143.00,87.88,0.00),v40,z0,tPen\WObj:=wPaper;
    MoveL Offs(pOrigin,144.20,88.12,0.00),v40,z0,tPen\WObj:=wPaper;
    MoveL Offs(pOrigin,144.20,88.12,0.00),v40,z0,tPen\WObj:=wPaper;
    MoveL Offs(pOrigin,146.15,88.28,0.00),v40,fine,tPen\WObj:=wPaper;
    MoveL Offs(pOrigin,146.15,88.28,6.00),v60,z5,tPen\WObj:=wPaper;
    MoveL Offs(pOrigin,147.35,86.93,6.00),vTravel,z5,tPen\WObj:=wPaper;
    MoveL Offs(pOrigin,147.35,86.93,0.00),v60,z0,tPen\WObj:=wPaper;
    MoveL Offs(pOrigin,147.50,86.62,0.00),v40,z0,tPen\WObj:=wPaper;
    MoveL Offs(pOrigin,147.05,86.32,0.00),v40,z0,tPen\WObj:=wPaper;
    MoveL Offs(pOrigin,147.50,85.72,0.00),v40,z0,tPen\WObj:=wPaper;
    MoveL Offs(pOrigin,147.50,85.72,0.00),v40,z0,tPen\WObj:=wPaper;
    MoveL Offs(pOrigin,147.05,85.18,0.00),v40,z0,tPen\WObj:=wPaper;
    MoveL Offs(pOrigin,144.20,88.12,0.00),v40,fine,tPen\WObj:=wPaper;
  ENDPROC

  PROC DrawPart9()
    MoveL Offs(pOrigin,144.20,88.12,6.00),v60,z5,tPen\WObj:=wPaper;
    MoveL Offs(pOrigin,142.40,87.22,6.00),vTravel,z5,tPen\WObj:=wPaper;
    MoveL Offs(pOrigin,142.40,87.22,0.00),v60,z0,tPen\WObj:=wPaper;
    MoveL Offs(pOrigin,139.70,89.82,0.00),v40,z0,tPen\WObj:=wPaper;
    MoveL Offs(pOrigin,139.25,89.88,0.00),v40,z0,tPen\WObj:=wPaper;
    MoveL Offs(pOrigin,138.35,89.03,0.00),v40,z0,tPen\WObj:=wPaper;
    MoveL Offs(pOrigin,138.35,89.03,0.00),v40,z0,tPen\WObj:=wPaper;
    MoveL Offs(pOrigin,141.95,85.43,0.00),v40,fine,tPen\WObj:=wPaper;
    MoveL Offs(pOrigin,141.95,85.43,6.00),v60,z5,tPen\WObj:=wPaper;
    MoveL Offs(pOrigin,141.50,84.07,6.00),vTravel,z5,tPen\WObj:=wPaper;
    MoveL Offs(pOrigin,141.50,84.07,0.00),v60,z0,tPen\WObj:=wPaper;
    MoveL Offs(pOrigin,137.30,87.97,0.00),v40,z0,tPen\WObj:=wPaper;
    MoveL Offs(pOrigin,137.30,87.97,0.00),v40,z0,tPen\WObj:=wPaper;
    MoveL Offs(pOrigin,137.45,89.18,0.00),v40,z0,tPen\WObj:=wPaper;
    MoveL Offs(pOrigin,137.45,89.18,0.00),v40,z0,tPen\WObj:=wPaper;
    MoveL Offs(pOrigin,138.35,90.18,0.00),v40,z0,tPen\WObj:=wPaper;
    MoveL Offs(pOrigin,139.10,89.93,0.00),v40,z0,tPen\WObj:=wPaper;
    MoveL Offs(pOrigin,139.10,89.93,0.00),v40,z0,tPen\WObj:=wPaper;
    MoveL Offs(pOrigin,138.35,89.03,0.00),v40,z0,tPen\WObj:=wPaper;
    MoveL Offs(pOrigin,138.35,89.03,0.00),v40,z0,tPen\WObj:=wPaper;
    MoveL Offs(pOrigin,137.45,89.18,0.00),v40,z0,tPen\WObj:=wPaper;
    MoveL Offs(pOrigin,137.30,89.18,0.00),v40,z0,tPen\WObj:=wPaper;
    MoveL Offs(pOrigin,135.80,89.28,0.00),v40,z0,tPen\WObj:=wPaper;
    MoveL Offs(pOrigin,135.05,87.22,0.00),v40,z0,tPen\WObj:=wPaper;
    MoveL Offs(pOrigin,135.25,86.47,0.00),v40,z0,tPen\WObj:=wPaper;
    MoveL Offs(pOrigin,136.40,85.57,0.00),v40,z0,tPen\WObj:=wPaper;
    MoveL Offs(pOrigin,136.40,85.57,0.00),v40,z0,tPen\WObj:=wPaper;
    MoveL Offs(pOrigin,136.40,86.93,0.00),v40,z0,tPen\WObj:=wPaper;
    MoveL Offs(pOrigin,136.70,87.53,0.00),v40,z0,tPen\WObj:=wPaper;
    MoveL Offs(pOrigin,135.65,88.43,0.00),v40,fine,tPen\WObj:=wPaper;
    MoveL Offs(pOrigin,135.65,88.43,6.00),v60,z5,tPen\WObj:=wPaper;
    MoveL Offs(pOrigin,137.60,89.62,6.00),vTravel,z5,tPen\WObj:=wPaper;
    MoveL Offs(pOrigin,137.60,89.62,0.00),v60,z0,tPen\WObj:=wPaper;
    MoveL Offs(pOrigin,138.05,90.07,0.00),v40,z0,tPen\WObj:=wPaper;
    MoveL Offs(pOrigin,137.60,89.62,0.00),v40,fine,tPen\WObj:=wPaper;
    MoveL Offs(pOrigin,137.60,89.62,6.00),v60,z5,tPen\WObj:=wPaper;
    MoveL Offs(pOrigin,136.40,85.57,6.00),vTravel,z5,tPen\WObj:=wPaper;
    MoveL Offs(pOrigin,136.40,85.57,0.00),v60,z0,tPen\WObj:=wPaper;
    MoveL Offs(pOrigin,139.55,82.43,0.00),v40,z0,tPen\WObj:=wPaper;
    MoveL Offs(pOrigin,139.10,81.38,0.00),v40,z0,tPen\WObj:=wPaper;
    MoveL Offs(pOrigin,137.30,77.18,0.00),v40,z0,tPen\WObj:=wPaper;
    MoveL Offs(pOrigin,137.45,76.43,0.00),v40,z0,tPen\WObj:=wPaper;
    MoveL Offs(pOrigin,137.00,74.93,0.00),v40,z0,tPen\WObj:=wPaper;
    MoveL Offs(pOrigin,137.00,74.93,0.00),v40,z0,tPen\WObj:=wPaper;
    MoveL Offs(pOrigin,137.30,74.62,0.00),v40,z0,tPen\WObj:=wPaper;
    MoveL Offs(pOrigin,137.15,73.12,0.00),v40,z0,tPen\WObj:=wPaper;
    MoveL Offs(pOrigin,137.15,73.12,0.00),v40,z0,tPen\WObj:=wPaper;
    MoveL Offs(pOrigin,142.70,67.88,0.00),v40,z0,tPen\WObj:=wPaper;
    MoveL Offs(pOrigin,142.70,67.88,0.00),v40,z0,tPen\WObj:=wPaper;
    MoveL Offs(pOrigin,143.15,69.07,0.00),v40,z0,tPen\WObj:=wPaper;
    MoveL Offs(pOrigin,143.15,69.07,0.00),v40,z0,tPen\WObj:=wPaper;
    MoveL Offs(pOrigin,144.50,70.12,0.00),v40,fine,tPen\WObj:=wPaper;
    MoveL Offs(pOrigin,144.50,70.12,6.00),v60,z5,tPen\WObj:=wPaper;
    MoveL Offs(pOrigin,142.70,67.88,6.00),vTravel,z5,tPen\WObj:=wPaper;
    MoveL Offs(pOrigin,142.70,67.88,0.00),v60,z0,tPen\WObj:=wPaper;
    MoveL Offs(pOrigin,141.30,63.22,0.00),v40,z0,tPen\WObj:=wPaper;
    MoveL Offs(pOrigin,140.75,62.62,0.00),v40,fine,tPen\WObj:=wPaper;
    MoveL Offs(pOrigin,140.75,62.62,6.00),v60,z5,tPen\WObj:=wPaper;
    MoveL Offs(pOrigin,141.20,58.58,6.00),vTravel,z5,tPen\WObj:=wPaper;
    MoveL Offs(pOrigin,141.20,58.58,0.00),v60,z0,tPen\WObj:=wPaper;
    MoveL Offs(pOrigin,141.05,59.33,0.00),v40,z0,tPen\WObj:=wPaper;
    MoveL Offs(pOrigin,146.45,64.72,0.00),v40,z0,tPen\WObj:=wPaper;
    MoveL Offs(pOrigin,147.05,65.78,0.00),v40,z0,tPen\WObj:=wPaper;
    MoveL Offs(pOrigin,147.05,65.78,0.00),v40,z0,tPen\WObj:=wPaper;
    MoveL Offs(pOrigin,151.55,61.42,0.00),v40,z0,tPen\WObj:=wPaper;
    MoveL Offs(pOrigin,151.55,61.42,0.00),v40,z0,tPen\WObj:=wPaper;
    MoveL Offs(pOrigin,152.00,61.58,0.00),v40,z0,tPen\WObj:=wPaper;
    MoveL Offs(pOrigin,152.30,62.17,0.00),v40,z0,tPen\WObj:=wPaper;
    MoveL Offs(pOrigin,152.30,62.17,0.00),v40,z0,tPen\WObj:=wPaper;
    MoveL Offs(pOrigin,152.90,62.47,0.00),v40,z0,tPen\WObj:=wPaper;
    MoveL Offs(pOrigin,153.05,63.22,0.00),v40,z0,tPen\WObj:=wPaper;
    MoveL Offs(pOrigin,153.05,63.22,0.00),v40,z0,tPen\WObj:=wPaper;
    MoveL Offs(pOrigin,154.25,63.72,0.00),v40,z0,tPen\WObj:=wPaper;
    MoveL Offs(pOrigin,154.70,64.57,0.00),v40,z0,tPen\WObj:=wPaper;
    MoveL Offs(pOrigin,155.50,65.18,0.00),v40,z0,tPen\WObj:=wPaper;
    MoveL Offs(pOrigin,155.65,65.78,0.00),v40,z0,tPen\WObj:=wPaper;
    MoveL Offs(pOrigin,157.05,67.28,0.00),v40,z0,tPen\WObj:=wPaper;
    MoveL Offs(pOrigin,157.40,68.62,0.00),v40,z0,tPen\WObj:=wPaper;
    MoveL Offs(pOrigin,157.40,68.62,0.00),v40,z0,tPen\WObj:=wPaper;
    MoveL Offs(pOrigin,158.00,70.28,0.00),v40,fine,tPen\WObj:=wPaper;
    MoveL Offs(pOrigin,158.00,70.28,6.00),v60,z5,tPen\WObj:=wPaper;
    MoveL Offs(pOrigin,157.40,68.62,6.00),vTravel,z5,tPen\WObj:=wPaper;
    MoveL Offs(pOrigin,157.40,68.62,0.00),v60,z0,tPen\WObj:=wPaper;
    MoveL Offs(pOrigin,153.95,72.07,0.00),v40,z0,tPen\WObj:=wPaper;
    MoveL Offs(pOrigin,152.60,72.68,0.00),v40,z0,tPen\WObj:=wPaper;
    MoveL Offs(pOrigin,149.90,75.22,0.00),v40,fine,tPen\WObj:=wPaper;
    MoveL Offs(pOrigin,149.90,75.22,6.00),v60,z5,tPen\WObj:=wPaper;
    MoveL Offs(pOrigin,149.30,74.03,6.00),vTravel,z5,tPen\WObj:=wPaper;
    MoveL Offs(pOrigin,149.30,74.03,0.00),v60,z0,tPen\WObj:=wPaper;
    MoveL Offs(pOrigin,156.50,66.97,0.00),v40,fine,tPen\WObj:=wPaper;
    MoveL Offs(pOrigin,156.50,66.97,6.00),v60,z5,tPen\WObj:=wPaper;
    MoveL Offs(pOrigin,155.60,65.93,6.00),vTravel,z5,tPen\WObj:=wPaper;
    MoveL Offs(pOrigin,155.60,65.93,0.00),v60,z0,tPen\WObj:=wPaper;
    MoveL Offs(pOrigin,151.40,70.12,0.00),v40,z0,tPen\WObj:=wPaper;
    MoveL Offs(pOrigin,151.35,70.18,0.00),v40,z0,tPen\WObj:=wPaper;
    MoveL Offs(pOrigin,150.80,70.78,0.00),v40,z0,tPen\WObj:=wPaper;
    MoveL Offs(pOrigin,150.45,70.57,0.00),v40,z0,tPen\WObj:=wPaper;
    MoveL Offs(pOrigin,150.65,70.22,0.00),v40,z0,tPen\WObj:=wPaper;
    MoveL Offs(pOrigin,151.35,70.18,0.00),v40,fine,tPen\WObj:=wPaper;
    MoveL Offs(pOrigin,151.35,70.18,6.00),v60,z5,tPen\WObj:=wPaper;
    MoveL Offs(pOrigin,150.20,68.93,6.00),vTravel,z5,tPen\WObj:=wPaper;
    MoveL Offs(pOrigin,150.20,68.93,0.00),v60,z0,tPen\WObj:=wPaper;
    MoveL Offs(pOrigin,150.60,68.88,0.00),v40,z0,tPen\WObj:=wPaper;
    MoveL Offs(pOrigin,154.70,64.72,0.00),v40,fine,tPen\WObj:=wPaper;
    MoveL Offs(pOrigin,154.70,64.72,6.00),v60,z5,tPen\WObj:=wPaper;
    MoveL Offs(pOrigin,153.95,63.67,6.00),vTravel,z5,tPen\WObj:=wPaper;
    MoveL Offs(pOrigin,153.95,63.67,0.00),v60,z0,tPen\WObj:=wPaper;
    MoveL Offs(pOrigin,149.60,68.18,0.00),v40,z0,tPen\WObj:=wPaper;
    MoveL Offs(pOrigin,149.30,67.12,0.00),v40,z0,tPen\WObj:=wPaper;
    MoveL Offs(pOrigin,153.05,63.22,0.00),v40,fine,tPen\WObj:=wPaper;
    MoveL Offs(pOrigin,153.05,63.22,6.00),v60,z5,tPen\WObj:=wPaper;
    MoveL Offs(pOrigin,152.30,62.17,6.00),vTravel,z5,tPen\WObj:=wPaper;
    MoveL Offs(pOrigin,152.30,62.17,0.00),v60,z0,tPen\WObj:=wPaper;
    MoveL Offs(pOrigin,148.10,66.38,0.00),v40,z0,tPen\WObj:=wPaper;
    MoveL Offs(pOrigin,147.20,66.38,0.00),v40,fine,tPen\WObj:=wPaper;
    MoveL Offs(pOrigin,147.20,66.38,6.00),v60,z5,tPen\WObj:=wPaper;
    MoveL Offs(pOrigin,151.55,61.42,6.00),vTravel,z5,tPen\WObj:=wPaper;
    MoveL Offs(pOrigin,151.55,61.42,0.00),v60,z0,tPen\WObj:=wPaper;
    MoveL Offs(pOrigin,151.10,60.72,0.00),v40,z0,tPen\WObj:=wPaper;
    MoveL Offs(pOrigin,141.20,58.58,0.00),v40,fine,tPen\WObj:=wPaper;
  ENDPROC

  PROC DrawPart10()
    MoveL Offs(pOrigin,141.20,58.58,6.00),v60,z5,tPen\WObj:=wPaper;
    MoveL Offs(pOrigin,135.35,70.28,6.00),vTravel,z5,tPen\WObj:=wPaper;
    MoveL Offs(pOrigin,135.35,70.28,0.00),v60,z0,tPen\WObj:=wPaper;
    MoveL Offs(pOrigin,135.05,70.72,0.00),v40,z0,tPen\WObj:=wPaper;
    MoveL Offs(pOrigin,135.80,71.47,0.00),v40,z0,tPen\WObj:=wPaper;
    MoveL Offs(pOrigin,135.80,71.47,0.00),v40,z0,tPen\WObj:=wPaper;
    MoveL Offs(pOrigin,135.05,70.88,0.00),v40,z0,tPen\WObj:=wPaper;
    MoveL Offs(pOrigin,135.95,70.57,0.00),v40,z0,tPen\WObj:=wPaper;
    MoveL Offs(pOrigin,135.80,72.07,0.00),v40,z0,tPen\WObj:=wPaper;
    MoveL Offs(pOrigin,135.80,72.07,0.00),v40,z0,tPen\WObj:=wPaper;
    MoveL Offs(pOrigin,136.40,72.22,0.00),v40,z0,tPen\WObj:=wPaper;
    MoveL Offs(pOrigin,137.15,73.12,0.00),v40,fine,tPen\WObj:=wPaper;
    MoveL Offs(pOrigin,137.15,73.12,6.00),v60,z5,tPen\WObj:=wPaper;
    MoveL Offs(pOrigin,136.10,73.88,6.00),vTravel,z5,tPen\WObj:=wPaper;
    MoveL Offs(pOrigin,136.10,73.88,0.00),v60,z0,tPen\WObj:=wPaper;
    MoveL Offs(pOrigin,137.00,74.93,0.00),v40,z0,tPen\WObj:=wPaper;
    MoveL Offs(pOrigin,137.00,74.93,0.00),v40,z0,tPen\WObj:=wPaper;
    MoveL Offs(pOrigin,136.10,74.18,0.00),v40,z0,tPen\WObj:=wPaper;
    MoveL Offs(pOrigin,135.80,73.88,0.00),v40,z0,tPen\WObj:=wPaper;
    MoveL Offs(pOrigin,135.35,73.43,0.00),v40,z0,tPen\WObj:=wPaper;
    MoveL Offs(pOrigin,135.40,72.38,0.00),v40,z0,tPen\WObj:=wPaper;
    MoveL Offs(pOrigin,135.80,72.07,0.00),v40,fine,tPen\WObj:=wPaper;
    MoveL Offs(pOrigin,135.80,72.07,6.00),v60,z5,tPen\WObj:=wPaper;
    MoveL Offs(pOrigin,142.10,75.97,6.00),vTravel,z5,tPen\WObj:=wPaper;
    MoveL Offs(pOrigin,142.10,75.97,0.00),v60,z0,tPen\WObj:=wPaper;
    MoveL Offs(pOrigin,141.50,76.57,0.00),v40,z0,tPen\WObj:=wPaper;
    MoveL Offs(pOrigin,141.65,77.03,0.00),v40,z0,tPen\WObj:=wPaper;
    MoveL Offs(pOrigin,141.65,77.03,0.00),v40,z0,tPen\WObj:=wPaper;
    MoveL Offs(pOrigin,138.65,79.72,0.00),v40,fine,tPen\WObj:=wPaper;
    MoveL Offs(pOrigin,138.65,79.72,6.00),v60,z5,tPen\WObj:=wPaper;
    MoveL Offs(pOrigin,142.70,77.93,6.00),vTravel,z5,tPen\WObj:=wPaper;
    MoveL Offs(pOrigin,142.70,77.93,0.00),v60,z0,tPen\WObj:=wPaper;
    MoveL Offs(pOrigin,143.00,77.93,0.00),v40,z0,tPen\WObj:=wPaper;
    MoveL Offs(pOrigin,142.85,77.62,0.00),v40,z0,tPen\WObj:=wPaper;
    MoveL Offs(pOrigin,142.70,77.93,0.00),v40,z0,tPen\WObj:=wPaper;
    MoveL Offs(pOrigin,143.00,77.93,0.00),v40,z0,tPen\WObj:=wPaper;
    MoveL Offs(pOrigin,142.70,77.62,0.00),v40,z0,tPen\WObj:=wPaper;
    MoveL Offs(pOrigin,142.70,77.93,0.00),v40,fine,tPen\WObj:=wPaper;
    MoveL Offs(pOrigin,142.70,77.93,6.00),v60,z5,tPen\WObj:=wPaper;
    MoveL Offs(pOrigin,145.70,76.28,6.00),vTravel,z5,tPen\WObj:=wPaper;
    MoveL Offs(pOrigin,145.70,76.28,0.00),v60,z0,tPen\WObj:=wPaper;
    MoveL Offs(pOrigin,145.75,75.68,0.00),v40,z0,tPen\WObj:=wPaper;
    MoveL Offs(pOrigin,146.75,75.22,0.00),v40,z0,tPen\WObj:=wPaper;
    MoveL Offs(pOrigin,147.85,74.03,0.00),v40,z0,tPen\WObj:=wPaper;
    MoveL Offs(pOrigin,146.60,73.88,0.00),v40,fine,tPen\WObj:=wPaper;
    MoveL Offs(pOrigin,146.60,73.88,6.00),v60,z5,tPen\WObj:=wPaper;
    MoveL Offs(pOrigin,159.65,93.07,6.00),vTravel,z5,tPen\WObj:=wPaper;
    MoveL Offs(pOrigin,159.65,93.07,0.00),v60,z0,tPen\WObj:=wPaper;
    MoveL Offs(pOrigin,152.75,95.47,0.00),v40,z0,tPen\WObj:=wPaper;
    MoveL Offs(pOrigin,146.30,97.03,0.00),v40,z0,tPen\WObj:=wPaper;
    MoveL Offs(pOrigin,143.90,99.38,0.00),v40,z0,tPen\WObj:=wPaper;
    MoveL Offs(pOrigin,143.90,99.38,0.00),v40,z0,tPen\WObj:=wPaper;
    MoveL Offs(pOrigin,145.25,103.72,0.00),v40,z0,tPen\WObj:=wPaper;
    MoveL Offs(pOrigin,145.30,104.78,0.00),v40,z0,tPen\WObj:=wPaper;
    MoveL Offs(pOrigin,146.60,105.82,0.00),v40,z0,tPen\WObj:=wPaper;
    MoveL Offs(pOrigin,147.05,106.72,0.00),v40,z0,tPen\WObj:=wPaper;
    MoveL Offs(pOrigin,147.05,106.72,0.00),v40,z0,tPen\WObj:=wPaper;
    MoveL Offs(pOrigin,147.65,107.18,0.00),v40,z0,tPen\WObj:=wPaper;
    MoveL Offs(pOrigin,147.80,108.07,0.00),v40,z0,tPen\WObj:=wPaper;
    MoveL Offs(pOrigin,147.80,108.07,0.00),v40,z0,tPen\WObj:=wPaper;
    MoveL Offs(pOrigin,138.65,116.93,0.00),v40,z0,tPen\WObj:=wPaper;
    MoveL Offs(pOrigin,138.95,117.82,0.00),v40,z0,tPen\WObj:=wPaper;
    MoveL Offs(pOrigin,142.55,114.38,0.00),v40,z0,tPen\WObj:=wPaper;
    MoveL Offs(pOrigin,143.45,113.97,0.00),v40,z0,tPen\WObj:=wPaper;
    MoveL Offs(pOrigin,149.70,114.07,0.00),v40,z0,tPen\WObj:=wPaper;
    MoveL Offs(pOrigin,150.05,115.72,0.00),v40,z0,tPen\WObj:=wPaper;
    MoveL Offs(pOrigin,148.85,120.38,0.00),v40,z0,tPen\WObj:=wPaper;
    MoveL Offs(pOrigin,142.70,122.38,0.00),v40,z0,tPen\WObj:=wPaper;
    MoveL Offs(pOrigin,139.25,119.03,0.00),v40,fine,tPen\WObj:=wPaper;
    MoveL Offs(pOrigin,139.25,119.03,6.00),v60,z5,tPen\WObj:=wPaper;
    MoveL Offs(pOrigin,142.55,122.47,6.00),vTravel,z5,tPen\WObj:=wPaper;
    MoveL Offs(pOrigin,142.55,122.47,0.00),v60,z0,tPen\WObj:=wPaper;
    MoveL Offs(pOrigin,139.05,118.88,0.00),v40,z0,tPen\WObj:=wPaper;
    MoveL Offs(pOrigin,138.60,117.07,0.00),v40,z0,tPen\WObj:=wPaper;
    MoveL Offs(pOrigin,137.90,115.88,0.00),v40,z0,tPen\WObj:=wPaper;
    MoveL Offs(pOrigin,137.60,113.93,0.00),v40,z0,tPen\WObj:=wPaper;
    MoveL Offs(pOrigin,137.60,113.93,0.00),v40,z0,tPen\WObj:=wPaper;
    MoveL Offs(pOrigin,141.50,110.32,0.00),v40,z0,tPen\WObj:=wPaper;
    MoveL Offs(pOrigin,141.95,109.28,0.00),v40,z0,tPen\WObj:=wPaper;
    MoveL Offs(pOrigin,141.95,108.07,0.00),v40,z0,tPen\WObj:=wPaper;
    MoveL Offs(pOrigin,141.95,108.07,0.00),v40,z0,tPen\WObj:=wPaper;
    MoveL Offs(pOrigin,145.25,104.93,0.00),v40,fine,tPen\WObj:=wPaper;
    MoveL Offs(pOrigin,145.25,104.93,6.00),v60,z5,tPen\WObj:=wPaper;
    MoveL Offs(pOrigin,144.95,103.28,6.00),vTravel,z5,tPen\WObj:=wPaper;
    MoveL Offs(pOrigin,144.95,103.28,0.00),v60,z0,tPen\WObj:=wPaper;
    MoveL Offs(pOrigin,136.70,111.07,0.00),v40,z0,tPen\WObj:=wPaper;
    MoveL Offs(pOrigin,136.70,111.07,0.00),v40,z0,tPen\WObj:=wPaper;
    MoveL Offs(pOrigin,136.85,112.72,0.00),v40,z0,tPen\WObj:=wPaper;
    MoveL Offs(pOrigin,137.60,113.93,0.00),v40,fine,tPen\WObj:=wPaper;
    MoveL Offs(pOrigin,137.60,113.93,6.00),v60,z5,tPen\WObj:=wPaper;
    MoveL Offs(pOrigin,136.70,111.07,6.00),vTravel,z5,tPen\WObj:=wPaper;
    MoveL Offs(pOrigin,136.70,111.07,0.00),v60,z0,tPen\WObj:=wPaper;
    MoveL Offs(pOrigin,136.20,110.47,0.00),v40,z0,tPen\WObj:=wPaper;
    MoveL Offs(pOrigin,134.90,106.43,0.00),v40,fine,tPen\WObj:=wPaper;
    MoveL Offs(pOrigin,134.90,106.43,6.00),v60,z5,tPen\WObj:=wPaper;
    MoveL Offs(pOrigin,136.40,105.68,6.00),vTravel,z5,tPen\WObj:=wPaper;
    MoveL Offs(pOrigin,136.40,105.68,0.00),v60,z0,tPen\WObj:=wPaper;
    MoveL Offs(pOrigin,137.30,106.72,0.00),v40,z0,tPen\WObj:=wPaper;
    MoveL Offs(pOrigin,137.30,106.72,0.00),v40,z0,tPen\WObj:=wPaper;
    MoveL Offs(pOrigin,143.90,100.28,0.00),v40,fine,tPen\WObj:=wPaper;
    MoveL Offs(pOrigin,143.90,100.28,6.00),v60,z5,tPen\WObj:=wPaper;
    MoveL Offs(pOrigin,141.65,98.93,6.00),vTravel,z5,tPen\WObj:=wPaper;
    MoveL Offs(pOrigin,141.65,98.93,0.00),v60,z0,tPen\WObj:=wPaper;
    MoveL Offs(pOrigin,140.60,98.62,0.00),v40,fine,tPen\WObj:=wPaper;
    MoveL Offs(pOrigin,140.60,98.62,6.00),v60,z5,tPen\WObj:=wPaper;
    MoveL Offs(pOrigin,137.15,107.47,6.00),vTravel,z5,tPen\WObj:=wPaper;
    MoveL Offs(pOrigin,137.15,107.47,0.00),v60,z0,tPen\WObj:=wPaper;
    MoveL Offs(pOrigin,136.70,107.47,0.00),v40,z0,tPen\WObj:=wPaper;
    MoveL Offs(pOrigin,135.80,108.38,0.00),v40,fine,tPen\WObj:=wPaper;
    MoveL Offs(pOrigin,135.80,108.38,6.00),v60,z5,tPen\WObj:=wPaper;
    MoveL Offs(pOrigin,130.85,108.22,6.00),vTravel,z5,tPen\WObj:=wPaper;
    MoveL Offs(pOrigin,130.85,108.22,0.00),v60,z0,tPen\WObj:=wPaper;
    MoveL Offs(pOrigin,129.80,107.18,0.00),v40,fine,tPen\WObj:=wPaper;
    MoveL Offs(pOrigin,129.80,107.18,6.00),v60,z5,tPen\WObj:=wPaper;
    MoveL Offs(pOrigin,129.05,104.62,6.00),vTravel,z5,tPen\WObj:=wPaper;
    MoveL Offs(pOrigin,129.05,104.62,0.00),v60,z0,tPen\WObj:=wPaper;
    MoveL Offs(pOrigin,126.80,106.88,0.00),v40,fine,tPen\WObj:=wPaper;
    MoveL Offs(pOrigin,126.80,106.88,6.00),v60,z5,tPen\WObj:=wPaper;
    MoveL Offs(pOrigin,123.35,111.68,6.00),vTravel,z5,tPen\WObj:=wPaper;
    MoveL Offs(pOrigin,123.35,111.68,0.00),v60,z0,tPen\WObj:=wPaper;
  ENDPROC

  PROC DrawPart11()
    MoveL Offs(pOrigin,124.55,114.07,0.00),v40,fine,tPen\WObj:=wPaper;
    MoveL Offs(pOrigin,124.55,114.07,6.00),v60,z5,tPen\WObj:=wPaper;
    MoveL Offs(pOrigin,123.35,111.68,6.00),vTravel,z5,tPen\WObj:=wPaper;
    MoveL Offs(pOrigin,123.35,111.68,0.00),v60,z0,tPen\WObj:=wPaper;
    MoveL Offs(pOrigin,121.70,111.22,0.00),v40,fine,tPen\WObj:=wPaper;
    MoveL Offs(pOrigin,121.70,111.22,6.00),v60,z5,tPen\WObj:=wPaper;
    MoveL Offs(pOrigin,142.85,110.93,6.00),vTravel,z5,tPen\WObj:=wPaper;
    MoveL Offs(pOrigin,142.85,110.93,0.00),v60,z0,tPen\WObj:=wPaper;
    MoveL Offs(pOrigin,147.05,106.72,0.00),v40,fine,tPen\WObj:=wPaper;
    MoveL Offs(pOrigin,147.05,106.72,6.00),v60,z5,tPen\WObj:=wPaper;
    MoveL Offs(pOrigin,147.80,108.07,6.00),vTravel,z5,tPen\WObj:=wPaper;
    MoveL Offs(pOrigin,147.80,108.07,0.00),v60,z0,tPen\WObj:=wPaper;
    MoveL Offs(pOrigin,148.30,108.38,0.00),v40,z0,tPen\WObj:=wPaper;
    MoveL Offs(pOrigin,149.75,113.93,0.00),v40,fine,tPen\WObj:=wPaper;
    MoveL Offs(pOrigin,149.75,113.93,6.00),v60,z5,tPen\WObj:=wPaper;
    MoveL Offs(pOrigin,179.75,111.22,6.00),vTravel,z5,tPen\WObj:=wPaper;
    MoveL Offs(pOrigin,179.75,111.22,0.00),v60,z0,tPen\WObj:=wPaper;
    MoveL Offs(pOrigin,190.20,121.57,0.00),v40,z0,tPen\WObj:=wPaper;
    MoveL Offs(pOrigin,190.50,123.07,0.00),v40,z0,tPen\WObj:=wPaper;
    MoveL Offs(pOrigin,188.75,125.03,0.00),v40,z0,tPen\WObj:=wPaper;
    MoveL Offs(pOrigin,188.75,125.03,0.00),v40,z0,tPen\WObj:=wPaper;
    MoveL Offs(pOrigin,182.60,124.93,0.00),v40,z0,tPen\WObj:=wPaper;
    MoveL Offs(pOrigin,179.40,121.72,0.00),v40,z0,tPen\WObj:=wPaper;
    MoveL Offs(pOrigin,179.30,111.68,0.00),v40,z0,tPen\WObj:=wPaper;
    MoveL Offs(pOrigin,179.75,111.22,0.00),v40,z0,tPen\WObj:=wPaper;
    MoveL Offs(pOrigin,179.75,111.22,0.00),v40,z0,tPen\WObj:=wPaper;
    MoveL Offs(pOrigin,183.05,114.38,0.00),v40,z0,tPen\WObj:=wPaper;
    MoveL Offs(pOrigin,183.35,114.53,0.00),v40,z0,tPen\WObj:=wPaper;
    MoveL Offs(pOrigin,185.00,114.53,0.00),v40,z0,tPen\WObj:=wPaper;
    MoveL Offs(pOrigin,185.30,114.07,0.00),v40,z0,tPen\WObj:=wPaper;
    MoveL Offs(pOrigin,185.30,114.07,0.00),v40,z0,tPen\WObj:=wPaper;
    MoveL Offs(pOrigin,187.55,112.12,0.00),v40,z0,tPen\WObj:=wPaper;
    MoveL Offs(pOrigin,187.55,112.12,0.00),v40,z0,tPen\WObj:=wPaper;
    MoveL Offs(pOrigin,187.25,111.57,0.00),v40,z0,tPen\WObj:=wPaper;
    MoveL Offs(pOrigin,182.90,110.03,0.00),v40,z0,tPen\WObj:=wPaper;
    MoveL Offs(pOrigin,182.90,110.03,0.00),v40,z0,tPen\WObj:=wPaper;
    MoveL Offs(pOrigin,179.90,109.93,0.00),v40,z0,tPen\WObj:=wPaper;
    MoveL Offs(pOrigin,179.75,111.22,0.00),v40,fine,tPen\WObj:=wPaper;
    MoveL Offs(pOrigin,179.75,111.22,6.00),v60,z5,tPen\WObj:=wPaper;
    MoveL Offs(pOrigin,179.75,109.88,6.00),vTravel,z5,tPen\WObj:=wPaper;
    MoveL Offs(pOrigin,179.75,109.88,0.00),v60,z0,tPen\WObj:=wPaper;
    MoveL Offs(pOrigin,179.90,100.57,0.00),v40,z0,tPen\WObj:=wPaper;
    MoveL Offs(pOrigin,179.90,100.57,0.00),v40,z0,tPen\WObj:=wPaper;
    MoveL Offs(pOrigin,185.90,106.72,0.00),v40,z0,tPen\WObj:=wPaper;
    MoveL Offs(pOrigin,182.90,110.03,0.00),v40,fine,tPen\WObj:=wPaper;
    MoveL Offs(pOrigin,182.90,110.03,6.00),v60,z5,tPen\WObj:=wPaper;
    MoveL Offs(pOrigin,185.30,110.62,6.00),vTravel,z5,tPen\WObj:=wPaper;
    MoveL Offs(pOrigin,185.30,110.62,0.00),v60,z0,tPen\WObj:=wPaper;
    MoveL Offs(pOrigin,188.15,107.62,0.00),v40,z0,tPen\WObj:=wPaper;
    MoveL Offs(pOrigin,188.75,107.47,0.00),v40,z0,tPen\WObj:=wPaper;
    MoveL Offs(pOrigin,188.75,107.47,0.00),v40,z0,tPen\WObj:=wPaper;
    MoveL Offs(pOrigin,189.20,108.53,0.00),v40,fine,tPen\WObj:=wPaper;
    MoveL Offs(pOrigin,189.20,108.53,6.00),v60,z5,tPen\WObj:=wPaper;
    MoveL Offs(pOrigin,188.75,106.72,6.00),vTravel,z5,tPen\WObj:=wPaper;
    MoveL Offs(pOrigin,188.75,106.72,0.00),v60,z0,tPen\WObj:=wPaper;
    MoveL Offs(pOrigin,187.85,105.68,0.00),v40,fine,tPen\WObj:=wPaper;
    MoveL Offs(pOrigin,187.85,105.68,6.00),v60,z5,tPen\WObj:=wPaper;
    MoveL Offs(pOrigin,188.75,106.72,6.00),vTravel,z5,tPen\WObj:=wPaper;
    MoveL Offs(pOrigin,188.75,106.72,0.00),v60,z0,tPen\WObj:=wPaper;
    MoveL Offs(pOrigin,193.10,102.68,0.00),v40,z0,tPen\WObj:=wPaper;
    MoveL Offs(pOrigin,193.10,102.68,0.00),v40,z0,tPen\WObj:=wPaper;
    MoveL Offs(pOrigin,193.05,101.62,0.00),v40,z0,tPen\WObj:=wPaper;
    MoveL Offs(pOrigin,191.90,100.82,0.00),v40,z0,tPen\WObj:=wPaper;
    MoveL Offs(pOrigin,191.80,100.43,0.00),v40,z0,tPen\WObj:=wPaper;
    MoveL Offs(pOrigin,195.95,96.38,0.00),v40,z0,tPen\WObj:=wPaper;
    MoveL Offs(pOrigin,195.95,96.38,0.00),v40,z0,tPen\WObj:=wPaper;
    MoveL Offs(pOrigin,196.85,96.97,0.00),v40,z0,tPen\WObj:=wPaper;
    MoveL Offs(pOrigin,197.15,96.68,0.00),v40,z0,tPen\WObj:=wPaper;
    MoveL Offs(pOrigin,196.40,95.78,0.00),v40,z0,tPen\WObj:=wPaper;
    MoveL Offs(pOrigin,196.40,95.78,0.00),v40,z0,tPen\WObj:=wPaper;
    MoveL Offs(pOrigin,197.30,95.18,0.00),v40,z0,tPen\WObj:=wPaper;
    MoveL Offs(pOrigin,197.30,95.18,0.00),v40,z0,tPen\WObj:=wPaper;
    MoveL Offs(pOrigin,197.25,94.12,0.00),v40,z0,tPen\WObj:=wPaper;
    MoveL Offs(pOrigin,196.10,93.97,0.00),v40,z0,tPen\WObj:=wPaper;
    MoveL Offs(pOrigin,196.10,93.97,0.00),v40,z0,tPen\WObj:=wPaper;
    MoveL Offs(pOrigin,195.35,93.38,0.00),v40,z0,tPen\WObj:=wPaper;
    MoveL Offs(pOrigin,194.30,93.22,0.00),v40,z0,tPen\WObj:=wPaper;
    MoveL Offs(pOrigin,194.00,93.53,0.00),v40,z0,tPen\WObj:=wPaper;
    MoveL Offs(pOrigin,194.00,93.53,0.00),v40,z0,tPen\WObj:=wPaper;
    MoveL Offs(pOrigin,192.50,93.68,0.00),v40,z0,tPen\WObj:=wPaper;
    MoveL Offs(pOrigin,188.30,98.03,0.00),v40,fine,tPen\WObj:=wPaper;
    MoveL Offs(pOrigin,188.30,98.03,6.00),v60,z5,tPen\WObj:=wPaper;
    MoveL Offs(pOrigin,189.95,98.62,6.00),vTravel,z5,tPen\WObj:=wPaper;
    MoveL Offs(pOrigin,189.95,98.62,0.00),v60,z0,tPen\WObj:=wPaper;
    MoveL Offs(pOrigin,194.60,94.12,0.00),v40,z0,tPen\WObj:=wPaper;
    MoveL Offs(pOrigin,195.05,94.72,0.00),v40,z0,tPen\WObj:=wPaper;
    MoveL Offs(pOrigin,194.90,95.28,0.00),v40,z0,tPen\WObj:=wPaper;
    MoveL Offs(pOrigin,194.15,95.47,0.00),v40,z0,tPen\WObj:=wPaper;
    MoveL Offs(pOrigin,190.70,98.93,0.00),v40,z0,tPen\WObj:=wPaper;
    MoveL Offs(pOrigin,190.70,98.93,0.00),v40,z0,tPen\WObj:=wPaper;
    MoveL Offs(pOrigin,190.75,99.97,0.00),v40,z0,tPen\WObj:=wPaper;
    MoveL Offs(pOrigin,191.55,100.57,0.00),v40,z0,tPen\WObj:=wPaper;
    MoveL Offs(pOrigin,185.90,106.43,0.00),v40,z0,tPen\WObj:=wPaper;
    MoveL Offs(pOrigin,185.30,105.82,0.00),v40,z0,tPen\WObj:=wPaper;
    MoveL Offs(pOrigin,179.90,100.57,0.00),v40,z0,tPen\WObj:=wPaper;
    MoveL Offs(pOrigin,179.90,100.57,0.00),v40,z0,tPen\WObj:=wPaper;
    MoveL Offs(pOrigin,180.35,99.38,0.00),v40,z0,tPen\WObj:=wPaper;
    MoveL Offs(pOrigin,180.35,99.38,0.00),v40,z0,tPen\WObj:=wPaper;
    MoveL Offs(pOrigin,185.45,104.32,0.00),v40,z0,tPen\WObj:=wPaper;
    MoveL Offs(pOrigin,186.65,104.07,0.00),v40,z0,tPen\WObj:=wPaper;
    MoveL Offs(pOrigin,190.70,100.12,0.00),v40,z0,tPen\WObj:=wPaper;
    MoveL Offs(pOrigin,190.70,98.93,0.00),v40,z0,tPen\WObj:=wPaper;
    MoveL Offs(pOrigin,188.75,98.53,0.00),v40,z0,tPen\WObj:=wPaper;
    MoveL Offs(pOrigin,188.00,98.03,0.00),v40,z0,tPen\WObj:=wPaper;
    MoveL Offs(pOrigin,181.40,98.03,0.00),v40,z0,tPen\WObj:=wPaper;
    MoveL Offs(pOrigin,180.50,98.78,0.00),v40,z0,tPen\WObj:=wPaper;
    MoveL Offs(pOrigin,180.35,99.38,0.00),v40,z0,tPen\WObj:=wPaper;
    MoveL Offs(pOrigin,180.35,99.38,0.00),v40,z0,tPen\WObj:=wPaper;
    MoveL Offs(pOrigin,185.30,104.18,0.00),v40,fine,tPen\WObj:=wPaper;
    MoveL Offs(pOrigin,185.30,104.18,6.00),v60,z5,tPen\WObj:=wPaper;
    MoveL Offs(pOrigin,193.10,102.68,6.00),vTravel,z5,tPen\WObj:=wPaper;
    MoveL Offs(pOrigin,193.10,102.68,0.00),v60,z0,tPen\WObj:=wPaper;
    MoveL Offs(pOrigin,193.75,103.57,0.00),v40,z0,tPen\WObj:=wPaper;
    MoveL Offs(pOrigin,194.60,106.72,0.00),v40,z0,tPen\WObj:=wPaper;
    MoveL Offs(pOrigin,194.60,106.72,0.00),v40,z0,tPen\WObj:=wPaper;
    MoveL Offs(pOrigin,193.40,108.07,0.00),v40,z0,tPen\WObj:=wPaper;
    MoveL Offs(pOrigin,193.40,108.07,0.00),v40,z0,tPen\WObj:=wPaper;
    MoveL Offs(pOrigin,193.40,109.88,0.00),v40,z0,tPen\WObj:=wPaper;
    MoveL Offs(pOrigin,192.80,110.62,0.00),v40,fine,tPen\WObj:=wPaper;
    MoveL Offs(pOrigin,192.80,110.62,6.00),v60,z5,tPen\WObj:=wPaper;
  ENDPROC

